# B&R Automation Studio project NAEUL004C00R13L518F00 (part 65)

#### Local.var
```iecst
(*2021-08-01*)
(**)
(*Local Action, State & Status*)
VAR
	eAct : eHermesAction := HermesActIdle;
	eStat : eHermesAction := HermesActIdle;
	eHermesAct : eHermesAction;
	eMcParamAct : eMcParamAction;
	eMainStatus : eFBStatus := Idle;
	eStatus : eFBStatus := Idle;
	eStatus1 : eFBStatus := Idle;
	eStatus2 : eFBStatus := Idle;
	eStatus3 : eFBStatus := Idle;
	udiStatus : UDINT := 0;
	udiStatus1 : UDINT := 0;
	udiStatus2 : UDINT := 0;
	udiStatus3 : UDINT := 0;
	udiStatus4 : UDINT := 0;
	udiStatus5 : UDINT;
	sStatTxt : STRING[200] := '';
	a_sStatText : ARRAY[0..50] OF STRING[200] := ['Idling','Background Starting Operations','Background Stopping Operations','Deleting Old Log File','Creating Directory','Writing Retain File','Reading Retain File','Saving Configuration',43('')];
END_VAR
(**)
(*Local Alarm*)
VAR
	tyAlmData : tyAlmDat;
	tyAlmData1 : tyAlmDat;
	tyAlmData2 : tyAlmDat;
	tyAlmData3 : tyAlmDat;
	tyAlmData4 : tyAlmDat;
	tyInfoData : tyAlmDat;
	tyInfoData1 : tyAlmDat;
	tyInfoData2 : tyAlmDat;
	tyInfoData3 : tyAlmDat;
	tyInfoData4 : tyAlmDat;
	a_tyAlmText : ARRAY[10000..10250] OF tyAlmTxt := [(sAlmText:='Invalid Ident While Creating Server',sRcyText:='Problem Occurred In The TCP/IP Connection. Check The Connection And Try To Reconnect.'),(sAlmText:='Setting Keep Alive Interval Time Error While Creating Server',sRcyText:='Unable To Establish Connection Between Machine. Check For Setting And Resume Operation.'),(sAlmText:='Setting Keep Alive Idle Time Error While Creating Server',sRcyText:='Unable To Establish Connection Between Machine. Check For Setting And Resume Operation.'),(sAlmText:='Setting Keep Alive Count Error While Creating Server',sRcyText:='Unable To Establish Connection Between Machine. Check For Setting And Resume Operation.'),(sAlmText:='Setting Keep Alive Error While Creating Server',sRcyText:='Unable To Establish Connection Between Machine. Check For Setting And Resume Operation.'),(sAlmText:='Setting Receive Buffer Error While Creating Server',sRcyText:='Unable To Establish Connection Between Machine. Check For Setting And Resume Operation.'),(sAlmText:='Setting Send Buffer Error While Creating Server',sRcyText:='Unable To Establish Connection Between Machine. Check For Setting And Resume Operation.'),(sAlmText:='Setting No Waiting Error While Creating Server',sRcyText:='Unable To Establish Connection Between Machine. Check For Setting And Resume Operation.'),(sAlmText:='TCP Open Port Error While Creating Server',sRcyText:='Problem Occurred In The TCP/IP Connection. Check The Connection And Try To Reconnect.'),(sAlmText:='Closing TCP Error While Creating Server',sRcyText:='Problem Occurred In The TCP/IP Connection. Check The Connection And Try To Reconnect.'),(sAlmText:='Invalid Ident While Listening Client',sRcyText:='There Was A Problem Connecting To The Server. The Server May Not Exist or It is Unavailable At This Time. Check The Connection and Try Again.'),(0),(sAlmText:='Supervisory Hermes Connection Lost',sRcyText:='There Was A Problem Connecting To The Server. The Server May Not Exist or It is Unavailable At This Time. Check The Connection and Try Again.'),(0),(sAlmText:='Invalid Ident While Receiving Data',sRcyText:='Problem Occurred In The TCP/IP Connection. Check The Connection And Try To Reconnect.'),(sAlmText:='TCP Receive Data Error While Receiving Data',sRcyText:='Problem Occurred In The TCP/IP Connection. Check The Connection And Try To Reconnect.'),(sAlmText:='Receive SetConfiguration While Supervisory In Not Connected State',sRcyText:='Receive Illegal Message.'),(sAlmText:='Receive GetConfiguration While Supervisory In Not Connected State',sRcyText:='Receive Illegal Message.'),(sAlmText:='Receive CurrConfiguration While Supervisory In Not Connected State',sRcyText:='Receive Illegal Message.'),(sAlmText:='Receive SendWorkOrderInfo While Supervisory In Not Connected State',sRcyText:='Receive Illegal Message.'),(sAlmText:='Receive QueryWorkOrderInfo While Supervisory In Not Connected State',sRcyText:='Receive Illegal Message.'),(sAlmText:='Receive BoardArrived While Supervisory In Not Connected State',sRcyText:='Receive Illegal Message.'),(sAlmText:='Receive BoardDeparted While Supervisory In Not Connected State',sRcyText:='Receive Illegal Message.'),2((0)),(sAlmText:='Receive BoardAvailable While Downstream In Service Description State',sRcyText:='Receive Illegal Message.'),(sAlmText:='Receive RevokeBoardAvailable While Downstream In Service Description State',sRcyText:='Receive Illegal Message.'),(sAlmText:='Receive ServiceDescription While Supervisory In Service Description State',sRcyText:='Receive Illegal Message.'),(sAlmText:='Receive SetConfiguration While Supervisory In Service Description State',sRcyText:='Receive Illegal Message.'),(sAlmText:='Receive GetConfiguration While Supervisory In Service Description State',sRcyText:='Receive Illegal Message.'),(sAlmText:='Receive CurrConfiguration While Supervisory In Service Description State',sRcyText:='Receive Illegal Message.'),(sAlmText:='Receive SendWorkOrderInfo While Supervisory In Service Description State',sRcyText:='Receive Illegal Message.'),(sAlmText:='Receive QueryWorkOrderInfo While Supervisory In Service Description State',sRcyText:='Receive Illegal Message.'),(sAlmText:='Receive BoardArrived While Supervisory In Service Description State',sRcyText:='Receive Illegal Message.'),(sAlmText:='Receive BoardDeparted While Supervisory In Service Description State',sRcyText:='Receive Illegal Message.'),4((0)),(sAlmText:='Receive ServiceDescription While Supervisory In Connected State',sRcyText:='Receive Illegal Message.'),(sAlmText:='Receive CurrConfiguration While Supervisory In Connected State',sRcyText:='Receive Illegal Message.'),(sAlmText:='Receive QueryWorkOrderInfo While Supervisory In Connected State',sRcyText:='Receive Illegal Message.'),(sAlmText:='Receive BoardArrived While Supervisory In Connected State',sRcyText:='Receive Illegal Message.'),(sAlmText:='Receive BoardDeparted While Supervisory In Connected State',sRcyText:='Receive Illegal Message.'),43((0)),(sAlmText:='SystemId Missing While Checking Service Description',sRcyText:='Missing Input Value For SystemId. Fill Up The Value And Resend.'),(sAlmText:='Version Missing While Checking Service Description',sRcyText:='Missing Input Value For Version. Fill Up The Value And Resend.'),(sAlmText:='SupportedFeatures Missing While Checking Service Description',sRcyText:='Missing Input Value For SupportedFeatures. Fill Up The Value And Resend.'),2((0)),(sAlmText:='NotificationCode Out Of Range While Checking Notification',sRcyText:='NotificationCode Does Not Fall Within The Expected Range.'),(sAlmText:='NotificationCode Missing While Checking Notification',sRcyText:='Missing Input Value For NotificationCode. Fill Up The Value And Resend.'),(sAlmText:='Severity Missing While Checking Notification',sRcyText:='Missing Input Value For Severity. Fill Up The Value And Resend.'),(sAlmText:='Description Missing While Checking Notification',sRcyText:='Missing Input Value For Description. Fill Up The Value And Resend.'),10((0)),(sAlmText:='Supervisory Service Description Interchange Time Out',sRcyText:='Timeout Expired Before Operation Completed. Reset And Resume Operation.'),4((0)),(sAlmText:='Get Directory Info Error While Deleting Old Log',sRcyText:='An Error Was Encountered While Getting Directory Info. Please Contact Nutek For A Possible Solution.'),(sAlmText:='Directory Read Error While Deleting Old Log',sRcyText:='An Error Was Encountered While Reading Directory. Please Contact Nutek For A Possible Solution.'),(sAlmText:='File Delete Error While Deleting Old Log',sRcyText:='An Error Was Encountered While Trying To Delete File. Please Contact Nutek For A Possible Solution.'),(sAlmText:='File Open Error While Reading Retain File',sRcyText:='An Error Was Encountered While Trying To Open File. Please Contact Nutek For A Possible Solution.'),(sAlmText:='File Read Error While Reading Retain File',sRcyText:='An Error Was Encountered While Trying To Read File. Please Contact Nutek For A Possible Solution.'),(sAlmText:='File Close Error While Reading Retain File',sRcyText:='An Error Was Encountered While Trying To Close File. Please Contact Nutek For A Possible Solution.'),(sAlmText:='File Open Error While Writting Retain File',sRcyText:='An Error Was Encountered While Trying To Open File. Please Contact Nutek For A Possible Solution.'),(sAlmText:='File Create Error While Writting Retain File',sRcyText:='An Error Was Encountered While Trying To Create File. Please Contact Nutek For A Possible Solution.'),(sAlmText:='File Write Error While Writting Retain File',sRcyText:='An Error Was Encountered While Trying To Write File. Please Contact Nutek For A Possible Solution.'),(sAlmText:='File Close Error While Writting Retain File',sRcyText:='An Error Was Encountered While Trying To Close File. Please Contact Nutek For A Possible Solution.'),(sAlmText:='Directory Does Not Exist While Writing Retain File',sRcyText:='The Directory Does Not Exist. Please Contact Nutek For A Possible Solution.'),(sAlmText:='Revoke Board Available Request To Send From Supervisory Hermes',sRcyText:='Sending Illegal Message.'),(sAlmText:='Stop Transport Request To Send From Supervisory Hermes',sRcyText:='Sending Illegal Message.'),(sAlmText:='Transport Finished Request To Send From Supervisory Hermes',sRcyText:='Sending Illegal Message.'),(sAlmText:='Board Available Request To Send From Supervisory Hermes',sRcyText:='Sending Illegal Message.'),6((0)),(sAlmText:='Check Alive Time Out',sRcyText:='Timeout Expired Before Operation Completed. Reset And Resume Operation.'),(sAlmText:='Waiting Check Alive Time Out',sRcyText:='Timeout Expired Before Operation Completed. Reset And Resume Operation.'),(sAlmText:='Check Alive Id Mismatch',sRcyText:='The Check Alive Id Value Does Not Match. Change The Value And Resend The Value.'),(sAlmText:='Machine Ready Request To Send From Supervisory Hermes',sRcyText:='Sending Illegal Message.'),(sAlmText:='Revoke Machine Ready Request To Send From Supervisory Hermes',sRcyText:='Sending Illegal Message.'),(sAlmText:='Start Transport Request To Send From Supervisory Hermes',sRcyText:='Sending Illegal Message.'),(sAlmText:='Set Configuration Request To Send From Supervisory Hermes',sRcyText:='Sending Illegal Message.'),(sAlmText:='Get Configuration Request To Send From Supervisory Hermes',sRcyText:='Sending Illegal Message.'),(sAlmText:='Current Configuration Request To Send From Supervisory Hermes',sRcyText:='Sending Illegal Message.'),(sAlmText:='Board Forecast Request To Send From Supervisory Hermes',sRcyText:='Sending Illegal Message.'),(sAlmText:='Query Board Info Request To Send From Supervisory Hermes',sRcyText:='Sending Illegal Message.'),(sAlmText:='Invalid Ident While Sending Data',sRcyText:='Invalid Ident Value.'),(sAlmText:='TCP Retry Send Data Error While Sending Data',sRcyText:='Problem Occurred In The TCP/IP Connection. Check The Connection And Try To Reconnect.'),(sAlmText:='TCP Send Data Error',sRcyText:='Problem Occurred In The TCP/IP Connection. Check The Connection And Try To Reconnect.'),(sAlmText:='Invalid Ident While Closing TCP',sRcyText:='Invalid Ident Value.'),(sAlmText:='Closing TCP Error',sRcyText:='Problem Occurred In The TCP/IP Connection. Check The Connection And Try To Reconnect.'),(sAlmText:='File Open Error While Writing Log',sRcyText:='An Error Was Encountered While Trying To Open File. Please Contact Nutek For A Possible Solution.'),(sAlmText:='File Create Error While Writing Log',sRcyText:='An Error Was Encountered While Trying To Create File. Please Contact Nutek For A Possible Solution.'),(sAlmText:='Get File Info Error While Writing Log',sRcyText:='An Error Was Encountered While Getting File Info. Please Contact Nutek For A Possible Solution.'),(sAlmText:='File Write Error While Writing Log',sRcyText:='An Error Was Encountered While Trying To Write File. Please Contact Nutek For A Possible Solution.'),(sAlmText:='File Close Error While Writing Log',sRcyText:='An Error Was Encountered While Trying To Close File. Please Contact Nutek For A Possible Solution.'),(sAlmText:='Directory Does Not Exist While Writing Log',sRcyText:='The Directory Does Not Exist.Please Contact Nutek For A Possible Solution.'),(sAlmText:='Invalid Ident While Closing TCP',sRcyText:='Invalid Ident Value.'),(sAlmText:='Closing TCP Error',sRcyText:='Problem Occurred In The TCP/IP Connection. Check The Connection And Try To Reconnect.'),3((0)),(sAlmText:='Send Board Info Request To Send From Supervisory Hermes',sRcyText:='Sending Illegal Message.'),(sAlmText:='Query Work Order Info Request To Send From Supervisory Hermes',sRcyText:='Sending Illegal Message.'),(sAlmText:='Send Work Order Info Request To Send From Supervisory Hermes',sRcyText:='Sending Illegal Message.'),(sAlmText:='Board Arrived Request To Send From Supervisory Hermes',sRcyText:='Sending Illegal Message.'),(sAlmText:='Board Depated Request To Send From Supervisory Hermes',sRcyText:='Sending Illegal Message.'),(sAlmText:='QueryId Mismatch While Checking SendWorkOrderInfo and QueryWorkOrderInfo',sRcyText:='The QueryId Value Does Not Match. Change The Value And Resend The Value.'),(sAlmText:='QueryId Missing While Checking Send Work Order Info',sRcyText:='Missing Input Value For QueryId. Fill Up The Value And Resend.'),20((0)),(sAlmText:='File Open Error While Writing Config File',sRcyText:='An Error Was Encountered While Trying To Open File. Please Contact Nutek For A Possible Solution.'),(sAlmText:='File Create Error While Writing Config File',sRcyText:='An Error Was Encountered While Trying To Create File. Please Contact Nutek For A Possible Solution.'),(sAlmText:='File Write Error While Writing Config File',sRcyText:='An Error Was Encountered While Trying To Write File. Please Contact Nutek For A Possible Solution.'),(sAlmText:='File Close Error While Writing Config File',sRcyText:='An Error Was Encountered While Trying To Close File. Please Contact Nutek For A Possible Solution.'),(sAlmText:='Directory Does Not Exist While Writing Config File',sRcyText:='The Directory Does Not Exist. Please Contact Nutek For A Possible Solution.'),9((0)),(sAlmText:='File Open Error While Reading Loader Work Order Retain File',sRcyText:='An Error Was Encountered While Trying To Open File. Please Contact Nutek For A Possible Solution.'),(sAlmText:='File Read Error While Reading Loader Work Order Retain File',sRcyText:='An Error Was Encountered While Trying To Read File. Please Contact Nutek For A Possible Solution.'),(sAlmText:='File Close Error While Reading Loader Work Order Retain File',sRcyText:='An Error Was Encountered While Trying To Close File. Please Contact Nutek For A Possible Solution.'),(sAlmText:='File Open Error While WrittingLoader Work Order  Retain File',sRcyText:='An Error Was Encountered While Trying To Open File. Please Contact Nutek For A Possible Solution.'),(sAlmText:='File Create Error While Writting Loader Work Order Retain File',sRcyText:='An Error Was Encountered While Trying To Create File. Please Contact Nutek For A Possible Solution.'),(sAlmText:='File Write Error While Writting Loader Work Order Retain File',sRcyText:='An Error Was Encountered While Trying To Write File. Please Contact Nutek For A Possible Solution.'),(sAlmText:='File Close Error While Writting Loader Work Order  Retain File',sRcyText:='An Error Was Encountered While Trying To Close File. Please Contact Nutek For A Possible Solution.'),(sAlmText:='Directory Does Not Exist While Loader Work Order Writing Retain File',sRcyText:='The Directory Does Not Exist. Please Contact Nutek For A Possible Solution.'),(sAlmText:='File Open Error While Reading Loader Loaded Work Order Retain File',sRcyText:='An Error Was Encountered While Trying To Open File. Please Contact Nutek For A Possible Solution.'),(sAlmText:='File Read Error While Reading Loader Loaded Work Order Retain File',sRcyText:='An Error Was Encountered While Trying To Read File. Please Contact Nutek For A Possible Solution.'),(sAlmText:='File Close Error While Reading Loader Loaded Work Order Retain File',sRcyText:='An Error Was Encountered While Trying To Close File. Please Contact Nutek For A Possible Solution.'),(sAlmText:='File Open Error While Writting Loader Loaded Work Order Retain File',sRcyText:='An Error Was Encountered While Trying To Open File. Please Contact Nutek For A Possible Solution.'),(sAlmText:='File Create Error While Writting Loaded Work Order Retain File',sRcyText:='An Error Was Encountered While Trying To Create File. Please Contact Nutek For A Possible Solution.'),(sAlmText:='File Write Error While Writting Loader Loaded Work Order Retain File',sRcyText:='An Error Was Encountered While Trying To Write File. Please Contact Nutek For A Possible Solution.'),(sAlmText:='File Close Error While Writting Loader Loaded Work Order Retain File',sRcyText:='An Error Was Encountered While Trying To Close File. Please Contact Nutek For A Possible Solution.'),(sAlmText:='Directory Does Not Exist While Writing Loader Loaded Work Order Retain File',sRcyText:='The Directory Does Not Exist. Please Contact Nutek For A Possible Solution.'),(sAlmText:='File Open Error While Reading Bypass Work Order Retain File',sRcyText:='An Error Was Encountered While Trying To Open File. Please Contact Nutek For A Possible Solution.'),(sAlmText:='File Read Error While Reading Bypass  Work Order Retain File',sRcyText:='An Error Was Encountered While Trying To Read File. Please Contact Nutek For A Possible Solution.'),(sAlmText:='File Close Error While Reading Bypass Work Order Retain File',sRcyText:='An Error Was Encountered While Trying To Close File. Please Contact Nutek For A Possible Solution.'),(sAlmText:='File Open Error While Writting Bypass Work Order Retain File',sRcyText:='An Error Was Encountered While Trying To Open File. Please Contact Nutek For A Possible Solution.'),(sAlmText:='File Create Error While Writting Bypass  Work Order Retain File',sRcyText:='An Error Was Encountered While Trying To Create File. Please Contact Nutek For A Possible Solution.'),(sAlmText:='File Write Error While Writting Bypass  Work Order Retain File',sRcyText:='An Error Was Encountered While Trying To Write File. Please Contact Nutek For A Possible Solution.'),(sAlmText:='File Close Error While Writting Bypass  Work Order Retain File',sRcyText:='An Error Was Encountered While Trying To Close File. Please Contact Nutek For A Possible Solution.'),(sAlmText:='Directory Does Not Exist While Writing Bypass  Work Order Retain File',sRcyText:='The Directory Does Not Exist. Please Contact Nutek For A Possible Solution.'),0,26((0))];
END_VAR
(**)
(*Local Output*)
VAR
	bConnected : BOOL;
	bTest : BOOL;
	bTest1 : BOOL;
	bTest2 : BOOL;
	bHandshakeDone : BOOL;
	sInternalSnd : STRING[65535];
	bFileNotFound : BOOL := FALSE;
	bWriteConfig : BOOL := FALSE;
	bUpdateUIData : BOOL := FALSE;
END_VAR
(**)
(*Local Input*)
VAR
	udiRstErr : UDINT := 0;
	bPrep : BOOL := TRUE;
	bEn : BOOL := TRUE;
	bDis : BOOL := FALSE;
	tyParam : tyHermesSvyParam;
	sIPAddr : STRING[15] := '192.168.0.100';
	a_usiMacAddr : ARRAY[0..5] OF USINT := [6(0)];
	tyDTStructure : DTStructure := (year:=2020,month:=11,day:=05,wday:=05,hour:=21,minute:=28,second:=30,millisec:=123,microsec:=456);
	dtCurrDT : DATE_AND_TIME := DT#2019-02-23-12:30:50;
	sMcId : STRING[80] := '';
	sMagazineId : STRING[80] := '';
	iSlotId : INT;
	sBarcode : STRING[254] := '';
	eBoardTransfer1 : eHermesBoardTransfer := HermesTransferred;
	eBoardTransfer2 : eHermesBoardTransfer := HermesTransferred;
	eBoardTransfer3 : eHermesBoardTransfer := HermesTransferred;
	eBoardTransfer4 : eHermesBoardTransfer := HermesTransferred;
	sVersion : STRING[7] := '1.3';
	sWorkOrderId : STRING[80] := '';
	sBatchId : STRING[80] := '';
	sRecipeNm : STRING[254] := '';
	udiSndBffrSize : UDINT := 65536;
	udiRcvBffrSize : UDINT := 65536;
	udiAliveIdleTimeInSec : UDINT := 5;
	tConnTimeOut : TIME := T#30s;
	diTransferInTO : DINT := 30000;
	bNewBrdAvl : BOOL := FALSE;
	bOpsRun : BOOL := FALSE;
	udiFileKeepDay : UDINT := 30;
	sConfigFileName : STRING[80] := 'SvyHermes.dat';
	sProgNm : STRING[15] := 'SvyHermes';
	sRetainFileName : STRING[80] := 'WorkOrder.dat';
	sRetainFileName1 : STRING[80] := 'LoaderSendWorkOrder.dat';
	sRetainFileName2 : STRING[80] := 'LoaderLoadedSendWorkOrder.dat';
	sRetainFileName3 : STRING[80] := 'BypassSendWorkOrder.dat';
	bNtSettingsLoadDone : BOOL := TRUE;
	bSvyPrep : BOOL := FALSE;
	bSvyEn : BOOL := FALSE;
	sInfoMsg : STRING[200];
	sInfoMsg1 : STRING[200];
	sInfoMsg2 : STRING[200];
	sInfoMsg3 : STRING[200];
	sInfoMsg4 : STRING[200];
	bEndSen : BOOL := FALSE;
	tyHermesCurrConfiguration : tyHermesConfiguration;
	bQueryWorkOrderInfo : BOOL;
	bAcceptCondition : BOOL;
	bAllZonesEmpty : BOOL;
	bDeleteWorkOrder : BOOL;
	bFirstMcIntheLine : BOOL;
	bUSHermesStopTransportSnd1 : BOOL;
	bUSHermesStopTransportSnd2 : BOOL;
	bUSHermesStopTransportSnd3 : BOOL;
	bUSHermesStopTransportSnd4 : BOOL;
	bDSHermesTransportFinishedSnd1 : BOOL;
	bDSHermesTransportFinishedSnd2 : BOOL;
	bDSHermesTransportFinishedSnd3 : BOOL;
	bDSHermesTransportFinishedSnd4 : BOOL;
	tyUSHermesBoardArrivedData1 : tyHermesBoardAvailable;
	tyUSHermesBoardArrivedData2 : tyHermesBoardAvailable;
	tyUSHermesBoardArrivedData3 : tyHermesBoardAvailable;
	tyUSHermesBoardArrivedData4 : tyHermesBoardAvailable;
	tyDSHermesBoardDepartedData1 : tyHermesBoardAvailable;
	tyDSHermesBoardDepartedData2 : tyHermesBoardAvailable;
	tyDSHermesBoardDepartedData3 : tyHermesBoardAvailable;
	tyDSHermesBoardDepartedData4 : tyHermesBoardAvailable;
	bInternalUse : BOOL;
	sInternalRcv : STRING[65535];
END_VAR
(**)
(*Local*)
VAR
	bRstErr : BOOL;
	udiRstErrOld : UDINT;
	bInitDone : BOOL;
	bInitialDone : BOOL;
	bRun : BOOL;
	bStop : BOOL;
	bRstConnection : BOOL;
	bRstState : BOOL;
	bRcvWorkOrderInfo1 : BOOL;
	bRcvWorkOrderInfo2 : BOOL;
	bRcvWorkOrderInfo3 : BOOL;
	bRcvBypassWorkOrderInfo2 : BOOL;
	bRstWorkOrderInfo : BOOL;
	bFoundIndexUS1 : BOOL;
	bFoundIndexUS2 : BOOL;
	bFoundIndexUS3 : BOOL;
	bFoundIndexUS4 : BOOL;
	bFoundIndexDS1 : BOOL;
	bFoundIndexDS2 : BOOL;
	bFoundIndexDS3 : BOOL;
	bFoundIndexDS4 : BOOL;
	udiFoundIndexUS1 : UDINT;
	udiFoundIndexUS2 : UDINT;
	udiFoundIndexUS3 : UDINT;
	udiFoundIndexUS4 : UDINT;
	udiFoundIndexDS1 : UDINT;
	udiFoundIndexDS2 : UDINT;
	udiFoundIndexDS3 : UDINT;
	udiFoundIndexDS4 : UDINT;
	k : UDINT := 0;
	kk : UDINT := 0;
	j : INT := 1;
	jj : INT := 2;
	jjj : INT := 3;
	jjjj : INT := 4;
	udiSvrIdent : UDINT;
	udiClntIdent : UDINT;
	udiClntIdentExtra : UDINT;
	udiXMLTableWriteIdx : UDINT;
	udiMsgSendBffr : UDINT;
	udiSndMsgLen : UDINT;
	sSnd : STRING[65535];
	sRcv : STRING[65535];
	a_tyXMLTableDataRcv : ARRAY[0..200] OF tyXMLTableDat;
	a_tyXMLTableDataSnd : ARRAY[0..200] OF tyXMLTableDat;
	a_eMsgSend : ARRAY[0..50] OF eHermesMsgType;
	tyMsgTypeRcv : tyHermesMsgType;
	tyCheckAliveSnd : tyHermesCheckAlive;
	tyCheckAlivePingSnd : tyHermesCheckAlive;
	tyCheckAlivePongSnd : tyHermesCheckAlive;
	tyCheckAliveRcv : tyHermesCheckAlive;
	tyCheckAlivePingRcv : tyHermesCheckAlive;
	tyCheckAlivePongRcv : tyHermesCheckAlive;
	tyServiceDescriptionRcv : tyHermesServiceDescription;
	tySServiceDescriptionSnd : tyHermesSServiceDescription;
	tySServiceDescriptionRcv : tyHermesSServiceDescription;
	tyNotificationSnd : tyHermesNotification;
	tyNotificationRcv : tyHermesNotification;
	tyBoardAvailableRcv : tyHermesBoardAvailable;
	tyMachineReady : tyHermesMachineReady;
	tyStartTransport : tyHermesStartTransport;
	tyStopTransport : tyHermesStopTransport;
	tyTransportFinished : tyHermesTransportFinished;
	tySetConfiguration : tyHermesSetConfiguration;
	tySetConfigurationRcv : tyHermesSetConfiguration;
	tySetConfigurationModified : tyHermesSetConfiguration;
	tyCurrentConfigurationRcv : tyHermesCurrentConfiguration;
	tyCurrentConfigurationSnd : tyHermesCurrentConfiguration;
	tyBoardForecast : tyHermesBoardForecast;
	tyBoardArrivedRcv : tyHermesBoardArrived;
	tyBoardArrived1 : tyHermesBoardArrived;
	tyBoardArrived2 : tyHermesBoardArrived;
	tyBoardArrived3 : tyHermesBoardArrived;
	tyBoardArrived4 : tyHermesBoardArrived;
	tyBoardDepartedRcv : tyHermesBoardDeparted;
	tyBoardDeparted1 : tyHermesBoardDeparted;
	tyBoardDeparted2 : tyHermesBoardDeparted;
	tyBoardDeparted3 : tyHermesBoardDeparted;
	tyBoardDeparted4 : tyHermesBoardDeparted;
	tyQueryBoardInfo : tyHermesQueryBoardInfo;
	tySendBoardInfo : tyHermesSendBoardInfo;
	tyQueryWorkOrderInfo : tyHermesQueryWorkOrderInfo; (*Query For Loader Mode*)
	tyQueryBypassWorkOrderInfo : tyHermesQueryWorkOrderInfo; (*Query For Bypass mode*)
	tyReplyWorkOrderInfo : tyHermesReplyWorkOrderInfo;
	tySendWorkOrderInfoAcc : tyHermesSendWorkOrderInfo;
	tySendBypassWorkOrderInfoAcc : tyHermesSendWorkOrderInfo;
	tySendWorkOrderInfoRcv : tyHermesSendWorkOrderInfo;
	tyDummySendWorkOrderInfoRcv : tyHermesSendWorkOrderInfo;
	tySendWorkOrderInfoNewAcc : tyHermesSendWorkOrderInfo;
	fbCreateSvr : fbTCPCreateSvr;
	fbListen : fbTCPListen;
	fbRcv : fbTCPRcv;
	fbSend : fbTCPSnd;
	fbCloseSvr : fbTCPClose;
	fbCloseClnt : fbTCPClose;
	fbParseXMLTable : fbHermesParseXMLTable;
	fbCheckAlive : fbHermesCheckAlive;
	fbCheckAliveSendPing : fbHermesCheckAliveSendPing;
	fbCheckAliveRcvPing : fbHermesCheckAliveRcvPing;
	fbSequenceSvy : fbHermesSequenceSvy;
	fbSequenceTO : fbHermesSequenceSvyTO;
	eStatOld : eHermesAction := HermesActIdle;
	tyParamOld : tyHermesSvyParam;
	udiLogCntr : UDINT := 1;
	udiWriteLogCntr : UDINT := 1;
	a_sLogList : ARRAY[1..10] OF STRING[65535];
	sDT : STRING[80];
	dtCurrDTTemp : DATE_AND_TIME;
	fbFileAppend1 : fbFileFullAppend;
	fbFileOldDel1 : fbFileOldDel;
	fbFileRead1 : fbFileFullRead;
	fbFileWrite1 : fbFileFullWrite;
	fbFileRead2 : fbFileFullRead;
	fbFileWrite2 : fbFileFullWrite;
	fbFileRead3 : fbFileFullRead;
	fbFileWrite3 : fbFileFullWrite;
	fbFileRead4 : fbFileFullRead;
	fbFileWrite4 : fbFileFullWrite;
	fbDelayTm : TON;
	fbDelayTm1 : TON;
	fbParseBrdAvlExternal : fbHermesParseXMLTable;
	tyDsInternalBoardDeparted : {REDUND_UNREPLICABLE} tyHermesBoardAvailable;
	rThickness : REAL;
	rConveyorSpeed : REAL;
	rTopClearanceHeight : REAL;
	rBottomClearanceHeight : REAL;
	rWeight : REAL;
	udiTargetAddress : UDINT := 0;
	udiTargetAddress1 : UDINT := 0;
	udiSizeAddress : UDINT := 0;
	udiSizeAddress1 : UDINT := 0;
	udiRetainDataAddr : UDINT;
	udiRetainDataLen : UDINT;
	udiLoaderRetainDataAddr0 : UDINT;
	udiLoaderRetainDataLen0 : UDINT;
	udiLoaderRetainDataAddr1 : UDINT;
	udiLoaderRetainDataLen1 : UDINT;
	udiBypassRetainDataAddr0 : UDINT;
	udiBypassRetainDataLen0 : UDINT;
	tyHermesBARcv : tyHermesBoardAvailable;
	tyHermesBFRcv : tyHermesBoardForecast;
	bOpsConvWaitForTopUpBrd : BOOL;
	diReqWidthInUM : DINT;
	diReqLoaderWidthInUM : DINT;
	iWriteLogStep : INT := 0;
	bDIPresentSen : BOOL;
	bUITopUpBrdRdy : BOOL;
	bOpsConvStepAllwTopUpBrd : BOOL;
	bOpsConvTopUpBrdReq : BOOL;
	bLinkStepStackMode : BOOL;
	udiModuleNum : UDINT := 6761;
	bTransportFinish1 : BOOL;
	bTransportFinish2 : BOOL;
	bTransportFinish3 : BOOL;
END_VAR
```

#### Act_Alarm.st
```iecst
(** 2021-08-01 **)
ACTION Act_Alarm: //General

	//Error
	IF EDGEPOS(eStatus = Error) THEN

		tyAlmData.sProgNm		:= p_sProgNm;
		tyAlmData.udiCode		:= udiStatus;
		tyAlmData.eSeverity		:= AlmSeverityError;
		tyAlmData.udiRunTime	:= tyAlmData.udiRunTime + 1;
		tyAlmData.bAlm			:= TRUE;
		tyAlmData.udiModuleNum  := udiModuleNum;
		g_sSvyHermesProgNm		:= p_sProgNm;
		//Get Error Message
		IF tyAlmData.udiCode < 10000 OR tyAlmData.udiCode > 10199 THEN
			tyAlmData.sAlmMsg	:= 'Unknown';
			tyAlmData.sRcyMsg	:= 'Unknown';
		ELSE
			tyAlmData.sAlmMsg	:= a_tyAlmText[tyAlmData.udiCode].sAlmText;
			tyAlmData.sRcyMsg	:= a_tyAlmText[tyAlmData.udiCode].sRcyText;
		END_IF

		sStatTxt	:= tyAlmData.sAlmMsg;

	ELSIF bRstErr AND (tyAlmData.udiCode <> 0) THEN

		tyAlmData.udiCode	:= 0;
		tyAlmData.eSeverity	:= AlmSeverityNA;
		tyAlmData.sAlmMsg	:= '';
		tyAlmData.sRcyMsg	:= '';
		tyAlmData.bAlm			:= FALSE;
		sStatTxt	:= a_sStatText[eStat];

	END_IF

END_ACTION
```

#### Act_Alarm1.st
```iecst
(** 2021-08-01 **)
ACTION Act_Alarm1:

	//Error
	IF EDGEPOS(eStatus1 = Error) THEN

		tyAlmData1.sProgNm		:= p_sProgNm;
		tyAlmData1.udiCode		:= udiStatus1;
		tyAlmData1.eSeverity	:= AlmSeverityError;
		tyAlmData1.udiRunTime	:= tyAlmData1.udiRunTime + 1;
		tyAlmData1.bAlm			:= TRUE;
		tyAlmData1.udiModuleNum  := udiModuleNum;
		g_sSvyHermesProgNm		:= p_sProgNm;
		//Get Error Message
		IF tyAlmData1.udiCode < 10000 OR tyAlmData1.udiCode > 10199 THEN
			tyAlmData1.sAlmMsg	:= 'Unknown';
			tyAlmData1.sRcyMsg	:= 'Unknown';
		ELSE
			tyAlmData1.sAlmMsg	:= a_tyAlmText[tyAlmData1.udiCode].sAlmText;
			tyAlmData1.sRcyMsg	:= a_tyAlmText[tyAlmData1.udiCode].sRcyText;
		END_IF

		sStatTxt	:= tyAlmData1.sAlmMsg;

	ELSIF bRstErr AND (tyAlmData1.udiCode <> 0) THEN

		tyAlmData1.udiCode		:= 0;
		tyAlmData1.eSeverity	:= AlmSeverityNA;
		tyAlmData1.sAlmMsg		:= '';
		tyAlmData1.sRcyMsg		:= '';
		tyAlmData1.bAlm			:= FALSE;
		sStatTxt	:= a_sStatText[eStat];

	END_IF

END_ACTION
```

#### Act_Alarm2.st
```iecst
(** 2021-08-01 **)
ACTION Act_Alarm2:

	//Error
	IF EDGEPOS(eStatus2 = Error) THEN

		tyAlmData2.sProgNm		:= p_sProgNm;
		tyAlmData2.udiCode		:= udiStatus2;
		tyAlmData2.eSeverity	:= AlmSeverityError;
		tyAlmData2.udiRunTime	:= tyAlmData2.udiRunTime + 1;
		tyAlmData2.bAlm			:= TRUE;
		tyAlmData2.udiModuleNum  := udiModuleNum;
		g_sSvyHermesProgNm		:= p_sProgNm;
		//Get Error Message
		IF tyAlmData2.udiCode < 10000 OR tyAlmData2.udiCode > 10199 THEN
			tyAlmData2.sAlmMsg	:= 'Unknown';
			tyAlmData2.sRcyMsg	:= 'Unknown';
		ELSE
			tyAlmData2.sAlmMsg	:= a_tyAlmText[tyAlmData2.udiCode].sAlmText;
			tyAlmData2.sRcyMsg	:= a_tyAlmText[tyAlmData2.udiCode].sRcyText;
		END_IF

		sStatTxt	:= tyAlmData2.sAlmMsg;

	ELSIF bRstErr AND (tyAlmData2.udiCode <> 0) THEN

		tyAlmData2.udiCode		:= 0;
		tyAlmData2.eSeverity	:= AlmSeverityNA;
		tyAlmData2.sAlmMsg		:= '';
		tyAlmData2.sRcyMsg		:= '';
		tyAlmData2.bAlm			:= FALSE;
		sStatTxt	:= a_sStatText[eStat];

	END_IF

END_ACTION
```

#### Act_Alarm3.st
```iecst
(** 2021-08-01 **)
ACTION Act_Alarm3: //fbFileAppend1 Error

	//Error
	IF EDGEPOS(eStatus3 = Error) THEN

		tyAlmData3.sProgNm		:= p_sProgNm;
		tyAlmData3.udiCode		:= udiStatus3;
		tyAlmData3.eSeverity	:= AlmSeverityError;
		tyAlmData3.udiRunTime	:= tyAlmData3.udiRunTime + 1;
		tyAlmData3.bAlm			:= TRUE;
		tyAlmData3.udiModuleNum  := udiModuleNum;
		g_sSvyHermesProgNm		:= p_sProgNm;
		//Get Error Message
		IF tyAlmData3.udiCode < 10000 OR tyAlmData3.udiCode > 10199 THEN
			tyAlmData3.sAlmMsg	:= 'Unknown';
			tyAlmData3.sRcyMsg	:= 'Unknown';
		ELSE
			tyAlmData3.sAlmMsg	:= a_tyAlmText[tyAlmData3.udiCode].sAlmText;
			tyAlmData3.sRcyMsg	:= a_tyAlmText[tyAlmData3.udiCode].sRcyText;
		END_IF

		sStatTxt	:= tyAlmData3.sAlmMsg;

	ELSIF bRstErr AND (tyAlmData3.udiCode <> 0) THEN

		tyAlmData3.udiCode		:= 0;
		tyAlmData3.eSeverity	:= AlmSeverityNA;
		tyAlmData3.sAlmMsg		:= '';
		tyAlmData3.sRcyMsg		:= '';
		tyAlmData3.bAlm			:= FALSE;
		sStatTxt	:= a_sStatText[eStat];

	END_IF

END_ACTION
```

#### Act_Alarm4.st
```iecst
(** 2021-08-01 **)
ACTION Act_Alarm4: //Not Connected Warning

	//Warning
	IF ((bConnected = FALSE) AND (p_bSvyEn)) THEN

		tyAlmData4.sProgNm		:= p_sProgNm;
		tyAlmData4.udiCode		:= udiStatus4;
		tyAlmData4.eSeverity	:= AlmSeverityWarning;
		tyAlmData4.udiRunTime	:= tyAlmData4.udiRunTime + 1;
		tyAlmData4.bWarning			:= TRUE;
		tyAlmData4.udiModuleNum  := udiModuleNum;
		g_sSvyHermesProgNm		:= p_sProgNm;
		//Get Warning Message
		IF tyAlmData4.udiCode < 10000 OR tyAlmData4.udiCode > 10199 THEN
			tyAlmData4.sAlmMsg	:= 'Unknown';
			tyAlmData4.sRcyMsg	:= 'Unknown';
		ELSE
			tyAlmData4.sAlmMsg	:= a_tyAlmText[tyAlmData4.udiCode].sAlmText;
			tyAlmData4.sRcyMsg	:= a_tyAlmText[tyAlmData4.udiCode].sRcyText;
		END_IF

		sStatTxt	:= tyAlmData4.sAlmMsg;

	ELSIF (bConnected AND (tyAlmData4.udiCode <> 0)) OR (p_bSvyEn = FALSE) THEN

		tyAlmData4.udiCode		:= 0;
		tyAlmData4.eSeverity	:= AlmSeverityNA;
		tyAlmData4.sAlmMsg		:= '';
		tyAlmData4.sRcyMsg		:= '';
		tyAlmData4.bWarning			:= FALSE;
		sStatTxt	:= a_sStatText[eStat];

	END_IF

END_ACTION
```

#### Act_Background.st
```iecst
(** 2021-08-01 **)
ACTION Act_Background:

	IF bRun = TRUE THEN
		IF udiSvrIdent = 0 THEN
			IF p_bInternalUse = FALSE THEN
				Act_Background_TCPCreateSvr;

				tyParamOld	:= p_tyParam;
			ELSE
				udiSvrIdent	:= 1;
			END_IF

		ELSE
			IF bRstConnection = FALSE THEN

				Act_Background_ChgConfig;

				IF udiClntIdent = 0 THEN
					IF p_bInternalUse = FALSE THEN
						Act_Background_TCPListen;
					ELSE
						udiClntIdent	:= 1;
					END_IF

				ELSE
					Act_Background_TCPRcv;

					Act_Background_NotificationRcv;

					Act_Background_IllegalMsg;
					Act_Background_ChkParamRcv;
					Act_Background_CmpParamRcv;
					Act_Background_UpdtConfig;

					IF bHandshakeDone = TRUE THEN
						IF (p_tyParam.tSndAlive <> T#0s) AND (p_tyParam.tRcvAlive <> T#0s) THEN
							IF tySServiceDescriptionRcv.tyData.tySupportedFeatures.bFeatureCheckAliveResponse = TRUE AND p_tyParam.bFeatureCheckAliveResponse = TRUE THEN
								Act_Background_ChkAliveSendPing;
								Act_Background_ChkAliveRcvPing;
							ELSE
								Act_Background_ChkAlive;
							END_IF
						ELSE
							fbCheckAlive(bEn := FALSE);
							fbCheckAliveSendPing(bEn := FALSE);
							fbCheckAliveRcvPing(bEn := FALSE);
						END_IF
					END_IF

					Act_Background_Sequence;
					Act_Background_SequenceTO;
					Act_Background_Err;

					IF tySServiceDescriptionRcv.tyAvl.tySupportedFeatures.bFeatureSendWorkOrderInfo = TRUE AND p_tyParam.bFeatureQueryWorkOrderInfo AND bHandshakeDone THEN
						Act_Background_QueryWorkOrderInfo;
					END_IF

					Act_Background_SendBoardArrivedLane1;
					Act_Background_SendBoardArrivedLane2;
					Act_Background_SendBoardArrivedLane3;
					Act_Background_SendBoardArrivedLane4;
					Act_Background_SendBoardDepartedLane1;
					Act_Background_SendBoardDepartedLane2;
					Act_Background_SendBoardDepartedLane3;
					Act_Background_SendBoardDepartedLane4;
					Act_Background_TCPSend;

					Act_Background_Log;

				END_IF

			ELSE
				IF udiClntIdent <> 0 THEN
					Act_Background_TCPCloseClnt;
				ELSE
					IF udiSvrIdent <> 0 THEN
						Act_Background_TCPCloseSvr;
					END_IF
				END_IF

			END_IF

			//Second Client Connected
			IF udiClntIdentExtra = 0 THEN

			ELSE

			END_IF

		END_IF

		Act_Background_Stop;

	END_IF

	IF EDGENEG(bRun) OR EDGENEG(udiSvrIdent = 0) THEN
		//Reset
		fbCreateSvr(bEn := FALSE);
	END_IF

	IF EDGENEG(bRun) OR EDGENEG(udiClntIdent = 0) THEN
		//Reset
		fbListen(bEn := FALSE);

		bConnected	:= bRun;
	END_IF

	IF EDGENEG(bRun) OR EDGENEG(udiSvrIdent <> 0) OR EDGENEG(udiClntIdent <> 0) THEN
		fbRcv(bEn := FALSE);
		fbSequenceSvy(bEn := FALSE);
		fbSequenceTO(bEn := FALSE);
		fbCheckAlive(bEn := FALSE);
		fbCheckAliveSendPing(bEn := FALSE);
		fbCheckAliveRcvPing(bEn := FALSE);
		fbSend(bEn := FALSE);

		fbFileAppend1(bEn := FALSE);
		iWriteLogStep	:= 0;

		bConnected		:= FALSE;
		bHandshakeDone	:= FALSE;
		bRstState		:= FALSE;

		memset(ADR(tyMsgTypeRcv) , 0 , SIZEOF(tyMsgTypeRcv));
		memset(ADR(a_eMsgSend) , 0 , SIZEOF(a_eMsgSend));
		udiMsgSendBffr	:= 0;
	END_IF

	IF EDGENEG(bRun) OR EDGENEG(udiSvrIdent <> 0) THEN
		bRstConnection	:= FALSE;
		fbCloseSvr(bEn := FALSE);
	END_IF

	IF EDGENEG(bRun) OR EDGENEG(udiClntIdent <> 0) THEN
		fbCloseClnt(bEn := FALSE);
	END_IF

	//Reset Error
	IF (eStatus1 = Error) AND bRstErr THEN
		eStatus1	:= Idle;
		udiStatus1	:= 0;

		fbCreateSvr(bEn := FALSE);
		fbListen(bEn := FALSE);
		fbRcv(bEn := FALSE);
		fbSequenceSvy(bEn := FALSE);
		fbSend(bEn := FALSE);
		fbCloseSvr(bEn := FALSE);
		fbCloseClnt(bEn := FALSE);
		fbCheckAlive(bEn := FALSE);
		fbCheckAliveSendPing(bEn := FALSE);
		fbCheckAliveRcvPing(bEn := FALSE);
		fbSequenceTO(bEn := FALSE);

		fbFileAppend1(bEn := FALSE);
		iWriteLogStep	:= 0;

		bConnected		:= FALSE;
		bHandshakeDone	:= FALSE;
		bRstConnection	:= FALSE;
		bRstState		:= FALSE;

		memset(ADR(tyMsgTypeRcv) , 0 , SIZEOF(tyMsgTypeRcv));
		memset(ADR(a_eMsgSend) , 0 , SIZEOF(a_eMsgSend));
		udiMsgSendBffr	:= 0;
	END_IF

	IF (eStatus2 = Error) AND bRstErr THEN
		eStatus2	:= Idle;
		udiStatus2	:= 0;

		fbSequenceTO(bEn := FALSE);

	END_IF

	IF (eStatus3 = Error) AND bRstErr THEN
		eStatus3	:= Idle;
		udiStatus3	:= 0;

		fbFileAppend1(bEn := FALSE);
		iWriteLogStep	:= 0;
	END_IF

END_ACTION
```

#### Act_Background_CmpParamRcv.st
```iecst
(** 2021-08-01 **)
ACTION Act_Background_CmpParamRcv:

	IF eStatus2 <> Error THEN

		IF tySServiceDescriptionRcv.tyAvl.tySupportedFeatures.bFeatureSendWorkOrderInfo = TRUE AND p_tyParam.bFeatureQueryWorkOrderInfo THEN
				                                                                          //ADD
			IF tyMsgTypeRcv.bSendWorkOrderInfo = TRUE AND (p_bQueryWorkOrderInfo OR tyQueryWorkOrderInfo.tyAvl.bQueryId) THEN
				udiStatus2	:= fHermesChkParamSWQW(tySendWorkOrderInfoRcv , tyQueryWorkOrderInfo);
				udiStatus5  := fHermesChkParamSWBQW(tySendWorkOrderInfoRcv , tyQueryBypassWorkOrderInfo);	          //ADD

				IF udiStatus2 <> 0 AND udiStatus5 <> 0 THEN
					eStatus2	:= Error;

					IF udiStatus2 = 2767 THEN
						udiStatus2	:= 10164;	//QueryId Mismatch While Checking SendWorkOrderId & QueryWorkOrderId
					ELSIF udiStatus5 = 2767  THEN
						udiStatus2	:= 10164;	//QueryId Mismatch While Checking SendWorkOrderId & QueryWorkOrderId
					ELSIF udiStatus2 = 2768 THEN
						udiStatus2	:= 10165;	//QueryId Missing While Checking SendWorkOrderId & QueryWorkOrderId
					ELSIF udiStatus5 = 2768 THEN
						udiStatus2	:= 10165;	//QueryId Missing While Checking SendWorkOrderId & QueryWorkOrderId
					END_IF

					fHermesAddOneMsgSend(ADR(a_eMsgSend) , ADR(udiMsgSendBffr) , HermesMsgTypeNotification);

					tyNotificationSnd.tyAvl.bSeverity			:= TRUE;
					tyNotificationSnd.tyAvl.bNotificationCode	:= TRUE;
					tyNotificationSnd.tyAvl.bDescription		:= TRUE;
					tyNotificationSnd.tyData.eSeverity			:= HermesSeverityError;
					tyNotificationSnd.tyData.iNotificationCode	:= UDINT_TO_INT(udiStatus2);
					tyNotificationSnd.tyData.sDescription		:= a_tyAlmText[udiStatus2].sAlmText;

					tyMsgTypeRcv.bSendWorkOrderInfo := FALSE; //reset, else latching
				END_IF
			END_IF
		END_IF
	END_IF

		END_ACTION
```

#### Act_Background_ProcessData.st
```iecst
(** 2021-08-01 **)
ACTION Act_Background_ProcessData:

	//Write Config into "Hermes"
	fbDelayTm(IN := bWriteConfig, PT := T#0.5S); //Small Delay 0.5s to let Hermes take the Data, before WriteConfig

	IF fbDelayTm.Q THEN

		eHermesAct := HermesActWriteConfig;
		eMcParamAct := McParamActWrite;

		IF p_eHermesStatus = Done AND p_eHermesStat = HermesActWriteConfig AND p_eMcParamStat = McParamActWrite AND p_eMcParamStatus = Done THEN

		eMcParamAct     := McParamActIdle;
	   	eHermesAct		:= HermesActIdle;
		bWriteConfig    := FALSE;
		bUpdateUIData   := TRUE;
		fbDelayTm(IN := FALSE);
		tyInfoData.sProgNm		:= p_sProgNm;
		tyInfoData.udiCode		:= 10000;
		tyInfoData.eSeverity	:= AlmSeverityInfo;
		tyInfoData.sAlmMsg		:= p_sInfoMsg;

	    ELSIF  (p_eHermesStatus = Error AND p_eHermesStat = HermesActWriteConfig) OR (p_eMcParamStat = McParamActWrite AND p_eMcParamStatus = Error)  THEN

			eMcParamAct     := McParamActIdle;
		    eHermesAct		:= HermesActIdle;
		    bWriteConfig    := FALSE;
		    bUpdateUIData   := FALSE;
			fbDelayTm(IN := FALSE);

			fHermesAddOneMsgSend(ADR(a_eMsgSend) , ADR(udiMsgSendBffr) , HermesMsgTypeNotification);

			udiStatus2 := 10199; //SetConfiguration Failed, Please Send Again
			tyNotificationSnd.tyAvl.bSeverity			:= TRUE;
			tyNotificationSnd.tyAvl.bNotificationCode	:= TRUE;
			tyNotificationSnd.tyAvl.bDescription		:= TRUE;
			tyNotificationSnd.tyData.eSeverity			:= HermesSeverityFatalError;
			tyNotificationSnd.tyData.iNotificationCode	:= UDINT_TO_INT(udiStatus2);
			tyNotificationSnd.tyData.sDescription		:= a_tyAlmText[udiStatus2].sAlmText;

		END_IF
	END_IF

	//Update UI
	IF bUpdateUIData THEN
		tyInfoData.sProgNm		:= p_sProgNm;
		tyInfoData.udiCode		:= 10000;
		tyInfoData.eSeverity	:= AlmSeverityInfo;
		tyInfoData.sAlmMsg		:= p_sInfoMsg;
	END_IF

	//Auto Reset
	fbDelayTm1(IN := bUpdateUIData , PT := T#2S); //Auto reset the Info Msg C0009 page. No need press.
	IF fbDelayTm1.Q = TRUE THEN

		//Clear Info Message
		tyInfoData.sProgNm		:= '';
		tyInfoData.udiCode		:= 0;
		tyInfoData.eSeverity	:= AlmSeverityNA;
		tyInfoData.sAlmMsg		:= '';

		bUpdateUIData  := FALSE;
		bFoundIndexUS1 := FALSE;
		bFoundIndexUS2 := FALSE;
		bFoundIndexUS3 := FALSE;
		bFoundIndexUS4 := FALSE;
		bFoundIndexDS1 := FALSE;
		bFoundIndexDS2 := FALSE;
		bFoundIndexDS3 := FALSE;
		bFoundIndexDS4 := FALSE;

		fbDelayTm1(IN := FALSE);
	END_IF

	//BatchId from Supervisory System
	sBatchId := tySendWorkOrderInfoAcc.tyData.sBatchId;

	//Retain sWorkOrderId for machine power cycle
	p_udiRetainDataAddr	:= ADR(sWorkOrderId);
	p_udiRetainDataLen	:= SIZEOF(sWorkOrderId);

	//Write Retain
//	IF EDGEPOS(bRcvWorkOrderInfo1) THEN
//    	sWorkOrderId := tySendWorkOrderInfoAcc.tyData.sWorkOrderId; //Receive from Svy
//		p_eAct := HermesActWriteRetain;

	IF EDGEPOS(bRetainNewAcc) THEN
    	sWorkOrderId := tySendWorkOrderInfoNewAcc.tyData.sWorkOrderId; //Receive from Svy
		p_eAct := HermesActWriteRetain;

	ELSIF EDGENEG(p_bSvyEn = TRUE) OR EDGENEG(p_bSvyPrep = TRUE) THEN
		sWorkOrderId := ''; //Empty if Supervisory Hermes disable
		p_eAct := HermesActWriteRetain;

	ELSIF EDGENEG(p_tyHermesConfiguration.tySvyParam.bFeatureQueryWorkOrderInfo = TRUE) THEN
		sWorkOrderId := ''; //Empty if no support
		p_eAct := HermesActWriteRetain;

	ELSIF EDGEPOS(p_bDeleteWorkOrder) THEN
		sWorkOrderId := ''; //Delete from UI
		tySendWorkOrderInfoNewAcc := tyDummySendWorkOrderInfoRcv;
		p_eAct := HermesActWriteRetain;
		p_bDeleteWorkOrder := FALSE;
	END_IF

	//Retain tySendWorkOrderInfoAcc (Loader Accept data)
	p_udiLoaderRetainDataAddr0	:= ADR(tySendWorkOrderInfoAcc);
	p_udiLoaderRetainDataLen0   := SIZEOF(tySendWorkOrderInfoAcc);

	//Retain tySendWorkOrderInfoNewAcc (Loader loaded Accept data)
	p_udiLoaderRetainDataAddr1	:= ADR(tySendWorkOrderInfoNewAcc);
	p_udiLoaderRetainDataLen1   := SIZEOF(tySendWorkOrderInfoNewAcc);

     //Retain tySendBypassWorkOrderInfoAcc (Bypass Accept data)
	p_udiBypassRetainDataAddr0	:= ADR(tySendBypassWorkOrderInfoAcc);
	p_udiBypassRetainDataLen0   := SIZEOF(tySendBypassWorkOrderInfoAcc);

	IF EDGEPOS (bRcvWorkOrderInfo1) THEN
		p_eAct := HermesActWriteRetainSendWO1;

	ELSIF EDGEPOS (bRetainNewAcc OR p_bDeleteWorkOrder) THEN
		p_eAct := HermesActWriteRetainSendWO2;

	ELSIF EDGEPOS (bRcvWorkBypassOrderInfo) THEN
		p_eAct := HermesActWriteRetainSendWO3;
	END_IF

	IF eStatus = Done AND eStat = HermesActWriteRetain THEN
		p_eAct		:= HermesActIdle;
	ELSIF eStatus = Done AND eStat = HermesActWriteRetainSendWO1 THEN
		p_eAct		:= HermesActIdle;
	ELSIF eStatus = Done AND eStat = HermesActWriteRetainSendWO2 THEN
		p_eAct		:= HermesActIdle;
	ELSIF eStatus = Done AND eStat = HermesActWriteRetainSendWO3 THEN
		p_eAct		:= HermesActIdle;
	END_IF

//	//Testing -> Read Retain
//	IF EDGEPOS(bTest) THEN
//		p_eAct := HermesActReadRetain;
//	END_IF
//
//	IF eStatus = Done AND eStat = HermesActReadRetain THEN
//		p_eAct		:= HermesActIdle;
//	END_IF

END_ACTION
```

#### Act_Background_QueryWorkOrderInfo.st
```iecst
(** 2021-08-01 **)
ACTION Act_Background_QueryWorkOrderInfo:

	IF eStatus2 <> Error THEN

//		IF EDGEPOS(p_bQueryWorkOrderInfo) AND p_bAcceptCondition THEN

//		IF (EDGEPOS((p_bSiemensMcModeChgPrep AND p_bOpsConvWaitForTopUpBrd OR (p_usiLinkProdRcpCurrRcpMcMod = 0 AND bQueryloaderWorkOrder = FALSE) AND bConnected AND p_bOpsRun) AND p_bQueryWorkOrderInfo = FALSE AND bManualQueryWO = FALSE(*AND p_bSiemensMcModeChgPrep = FALSE)*)  (*AND p_bAcceptCondition*) AND bReplyWorkOrderInfo= FALSE AND sWorkOrderId = ''))
//			 OR EDGEPOS (p_bQueryWorkOrderInfo) THEN        //Query For Loader           //ADD
		IF (EDGEPOS((p_bSiemensMcModeChgPrep AND (p_bOpsConvWaitForTopUpBrd OR p_usiLinkProdRcpCurrRcpMcMod = 0)  AND bQueryloaderWorkOrder = FALSE AND bConnected AND p_bOpsRun) AND p_bQueryWorkOrderInfo = FALSE AND bManualQueryWO = FALSE AND bReplyWorkOrderInfo= FALSE AND sWorkOrderId = ''))
			 OR EDGEPOS (p_bQueryWorkOrderInfo) THEN        //Query For Loader           //ADD

			fHermesAddOneMsgSend(ADR(a_eMsgSend) , ADR(udiMsgSendBffr) , HermesMsgTypeQueryWorkOrderInfo);

			fHermesGenerateUUID(ADR(tyQueryWorkOrderInfo.tyData.sQueryId) , p_tyDTStructure , pa_usiMacAddr); //Generate QueryID

			tyQueryWorkOrderInfo.tyData.sMachineId							:= p_sMcId;
			tyQueryWorkOrderInfo.tyData.sMagazineId							:= p_sMagazineId;
			tyQueryWorkOrderInfo.tyData.iSlotId								:= p_iSlotId;
			tyQueryWorkOrderInfo.tyData.sBarcode						    := p_sBarcode;

			tyQueryWorkOrderInfo.tyAvl.bQueryId							    := tyQueryWorkOrderInfo.tyData.sQueryId <> '';
			tyQueryWorkOrderInfo.tyAvl.bMachineId							:= tyQueryWorkOrderInfo.tyData.sMachineId <> '';
			tyQueryWorkOrderInfo.tyAvl.bMagazineId							:= tyQueryWorkOrderInfo.tyData.sMagazineId <> '';
			tyQueryWorkOrderInfo.tyAvl.bSlotId								:= tyQueryWorkOrderInfo.tyData.iSlotId <> 0;
			tyQueryWorkOrderInfo.tyAvl.bBarcode								:= tyQueryWorkOrderInfo.tyData.sBarcode <> '';

			bQueryloaderWorkOrder := TRUE;
			bRcvWorkOrderInfo1 := FALSE;                     //ADD
			bRcvWorkOrderInfo2 := FALSE;

		END_IF
		                                                                      //Reply Bypass Workorder
		IF EDGEPOS((p_bSiemensMcModeChgPrep AND bConnected AND p_bOpsRun) AND bReplyBypassWorkOrderInfo= FALSE AND p_bUSHermesUSRdy AND bNewIncomingBoard)  THEN        //Query For Bypass mode           //ADD

			fHermesAddOneMsgSend(ADR(a_eMsgSend) , ADR(udiMsgSendBffr) , HermesMsgTypeQueryBypassWOInfo);

			fHermesGenerateUUID(ADR(tyQueryBypassWorkOrderInfo.tyData.sQueryId) , p_tyDTStructure , pa_usiMacAddr); //Generate QueryID

			tyQueryBypassWorkOrderInfo.tyData.sMachineId							:= p_sMcId;
			tyQueryBypassWorkOrderInfo.tyData.sMagazineId							:= p_sMagazineId;
			tyQueryBypassWorkOrderInfo.tyData.iSlotId								:= p_iSlotId;
			tyQueryBypassWorkOrderInfo.tyData.sBarcode						        := sUSBarcode;

			tyQueryBypassWorkOrderInfo.tyAvl.bQueryId							    := tyQueryBypassWorkOrderInfo.tyData.sQueryId <> '';
			tyQueryBypassWorkOrderInfo.tyAvl.bMachineId						     	:= tyQueryBypassWorkOrderInfo.tyData.sMachineId <> '';
			tyQueryBypassWorkOrderInfo.tyAvl.bMagazineId							:= tyQueryBypassWorkOrderInfo.tyData.sMagazineId <> '';
			tyQueryBypassWorkOrderInfo.tyAvl.bSlotId								:= tyQueryBypassWorkOrderInfo.tyData.iSlotId <> 0;
			tyQueryBypassWorkOrderInfo.tyAvl.bBarcode								:= tyQueryBypassWorkOrderInfo.tyData.sBarcode <> '';

			bQueryBypassWorkOrder := TRUE;
			bRcvWorkBypassOrderInfo := FALSE;
			bRcvBypassWorkOrderInfo2 := FALSE;
			bRcvWorkOrderInfo3      :=FALSE;
		END_IF

		IF p_bQueryWorkOrderInfo AND p_bAcceptCondition =FALSE THEN
			bRstWorkOrderInfo := TRUE;
		END_IF

		IF tyMsgTypeRcv.bSendWorkOrderInfo THEN

//			IF p_bQueryWorkOrderInfo AND (udiStatus2 = 0) THEN //After CmpParamRcv
//			IF (p_bQueryWorkOrderInfo OR p_bOpsConvWaitForTopUpBrd) AND (udiStatus2 = 0) AND p_tyDI.bTopCoverSWSig THEN //After CmpParamRcv
			IF (p_bQueryWorkOrderInfo OR p_bSiemensMcModeChgPrep) AND (udiStatus2 = 0) THEN //After CmpParamRcv
				IF tySendWorkOrderInfoRcv.tyAvl.bWorkOrderId AND tySendWorkOrderInfoRcv.tyData.sWorkOrderId <> '' AND
				   tySendWorkOrderInfoRcv.tyData.rWidth >= 50.0 AND tySendWorkOrderInfoRcv.tyData.rWidth <= 460.0	(*AND p_bAcceptCondition*) THEN //Wait Accept Conditon On

					bRcvWorkOrderInfo1 := TRUE;
					bRetainNewAcc      := FALSE;                            //ADD
					bQueryloaderWorkOrder := FALSE;
					tySendWorkOrderInfoAcc := tySendWorkOrderInfoRcv;
					tyMsgTypeRcv.bSendWorkOrderInfo := FALSE;
					sWorkOrderId := tySendWorkOrderInfoAcc.tyData.sWorkOrderId;

				ELSIF (tySendWorkOrderInfoRcv.tyAvl.bWorkOrderId = FALSE) OR tySendWorkOrderInfoRcv.tyData.sWorkOrderId = '' OR
					tySendWorkOrderInfoRcv.tyData.rWidth < 50.0 OR tySendWorkOrderInfoRcv.tyData.rWidth > 460.0  THEN
					bRcvWorkOrderInfo2 := TRUE;
					tyMsgTypeRcv.bSendWorkOrderInfo := FALSE;
				END_IF

			ELSIF p_bSiemensMcModeChgPrep AND (udiStatus5 = 0) THEN
				IF tySendWorkOrderInfoRcv.tyAvl.bWorkOrderId AND (tySendWorkOrderInfoRcv.tyData.sWorkOrderId = p_tyUSBoardAvailableRcv.tyData.sWorkOrderId OR tySendWorkOrderInfoRcv.tyData.sWorkOrderId = p_tyUSBoardForecastRcv.tyData.sWorkOrderId) AND
					tySendWorkOrderInfoRcv.tyAvl.bBatchId AND (tySendWorkOrderInfoRcv.tyData.sBatchId = p_tyUSBoardAvailableRcv.tyData.sBatchId OR tySendWorkOrderInfoRcv.tyData.sBatchId = p_tyUSBoardForecastRcv.tyData.sBatchId) AND
					tySendWorkOrderInfoRcv.tyAvl.bWidth AND (tySendWorkOrderInfoRcv.tyData.rWidth = p_tyUSBoardAvailableRcv.tyData.rWidth OR tySendWorkOrderInfoRcv.tyData.rWidth = p_tyUSBoardForecastRcv.tyData.rWidth) AND
					tySendWorkOrderInfoRcv.tyData.rWidth >= 50.0 AND tySendWorkOrderInfoRcv.tyData.rWidth <= 460.0 THEN
					bRcvWorkBypassOrderInfo := TRUE;
					tySendBypassWorkOrderInfoAcc := tySendWorkOrderInfoRcv;
					tyMsgTypeRcv.bSendWorkOrderInfo := FALSE;
					bRcvWorkOrderInfo3      :=TRUE;
				ELSE
					bRcvBypassWorkOrderInfo2 := TRUE;
					tyMsgTypeRcv.bSendWorkOrderInfo := FALSE;
				END_IF

//			ELSIF p_bQueryWorkOrderInfo = FALSE  THEN
			ELSIF p_bQueryWorkOrderInfo = FALSE  AND p_bLinkDIPresentSen = FALSE AND ((udiStatus2 = 0) OR (udiStatus5 = 0)) THEN
				tyMsgTypeRcv.bSendWorkOrderInfo := FALSE;
			END_IF
		END_IF

		IF EDGEPOS (bRcvWorkOrderInfo1 = TRUE AND p_bAcceptCondition) THEN

			tyInfoData1.sProgNm		:= p_sProgNm;
			tyInfoData1.udiCode		:= 10000;
			tyInfoData1.eSeverity	:= AlmSeverityInfo;
			tyInfoData1.sAlmMsg		:= p_sInfoMsg1;

		ELSIF EDGEPOS( bRcvWorkOrderInfo2 = TRUE OR bRcvBypassWorkOrderInfo2) THEN

			tyInfoData2.sProgNm		:= p_sProgNm;
			tyInfoData2.udiCode		:= 10000;
			tyInfoData2.eSeverity	:= AlmSeverityInfo;
			tyInfoData2.sAlmMsg		:= p_sInfoMsg2;

//			bRcvWorkOrderInfo2      := FALSE;
//			bRcvBypassWorkOrderInfo2 := FALSE;

		ELSIF EDGEPOS (bRcvWorkOrderInfo1 = TRUE AND p_bAcceptCondition = FALSE) THEN
			tyInfoData4.sProgNm		:= p_sProgNm;
			tyInfoData4.udiCode		:= 10000;
			tyInfoData4.eSeverity	:= AlmSeverityInfo;
			tyInfoData4.sAlmMsg		:= p_sInfoMsg4;

		END_IF

		IF  bRstWorkOrderInfo = TRUE THEN

			tyInfoData3.sProgNm		:= p_sProgNm;
			tyInfoData3.udiCode		:= 10000;
			tyInfoData3.eSeverity	:= AlmSeverityInfo;
			tyInfoData3.sAlmMsg		:= p_sInfoMsg3;

		END_IF

		IF EDGEPOS (bRcvWorkOrderInfo1 OR bRcvWorkOrderInfo2) THEN                       //ReplyWorkOrderInfo for loader

			fHermesAddOneMsgSend(ADR(a_eMsgSend) , ADR(udiMsgSendBffr) , HermesMsgTypeReplyWorkOrderInfo);

			tyReplyWorkOrderInfo.tyData.sWorkOrderId					    := tySendWorkOrderInfoAcc.tyData.sWorkOrderId;
			tyReplyWorkOrderInfo.tyData.sBatchId					      	:= tySendWorkOrderInfoAcc.tyData.sBatchId;
		    IF p_bAcceptCondition AND bRcvWorkOrderInfo2 = FALSE AND p_usiLinkProdRcpCurrRcpMcMod =1  THEN
				tyReplyWorkOrderInfo.tyData.iStatus							    := 1;          //WorkOrder accepted
				bReplyWorkOrderInfo                                             := TRUE;
			ELSIF bRcvWorkOrderInfo2 THEN
				tyReplyWorkOrderInfo.tyData.iStatus							    := 0;         //WorkOrder Rejected
				bReplyWorkOrderInfo                                             := FALSE;
				bRcvWorkOrderInfo2                                              := FALSE;
			ELSE
				tyReplyWorkOrderInfo.tyData.iStatus							    := 2;          //WorkOrder accepted and queue
				bReplyWorkOrderInfo                                             := TRUE;
			END_IF

			tyReplyWorkOrderInfo.tyAvl.bWorkOrderId					:= tySendWorkOrderInfoAcc.tyData.sWorkOrderId <> '';
			tyReplyWorkOrderInfo.tyAvl.bBatchId                     := tySendWorkOrderInfoAcc.tyData.sBatchId <> '';
			tyReplyWorkOrderInfo.tyAvl.bStatus                      :=  TRUE;
		END_IF

		IF EDGEPOS (bRcvWorkOrderInfo3 OR bRcvBypassWorkOrderInfo2) THEN                       //ReplyWorkOrderInfo for Bypass
			fHermesAddOneMsgSend(ADR(a_eMsgSend) , ADR(udiMsgSendBffr) , HermesMsgTypeReplyWorkOrderInfo);

			tyReplyWorkOrderInfo.tyData.sWorkOrderId					    := tySendBypassWorkOrderInfoAcc.tyData.sWorkOrderId;
			tyReplyWorkOrderInfo.tyData.sBatchId					      	:= tySendBypassWorkOrderInfoAcc.tyData.sBatchId;

			IF p_bAcceptCondition AND p_usiLinkProdRcpCurrRcpMcMod =0 AND bRcvWorkOrderInfo3  THEN
				tyReplyWorkOrderInfo.tyData.iStatus							    := 1;          //WorkOrder accepted
				bReplyBypassWorkOrderInfo                                       := TRUE;
			ELSIF p_bAcceptCondition AND p_usiLinkProdRcpCurrRcpMcMod =1 AND bRcvWorkOrderInfo3 THEN
				tyReplyWorkOrderInfo.tyData.iStatus							    := 2;          //WorkOrder accepted and queue
				bReplyBypassWorkOrderInfo                                       := TRUE;
				bQueryBypassWorkOrder := FALSE;                                               //Add
			ELSIF bRcvBypassWorkOrderInfo2 THEN
				tyReplyWorkOrderInfo.tyData.iStatus							    := 0;          //WorkOrder Rejected
				bReplyBypassWorkOrderInfo                                       := TRUE;
				bRcvBypassWorkOrderInfo2                                        :=FALSE;
			END_IF
			tyReplyWorkOrderInfo.tyAvl.bWorkOrderId					:= tySendWorkOrderInfoAcc.tyData.sWorkOrderId <> '';
			tyReplyWorkOrderInfo.tyAvl.bBatchId                     := tySendWorkOrderInfoAcc.tyData.sBatchId <> '';
			tyReplyWorkOrderInfo.tyAvl.bStatus                      :=  TRUE;
		END_IF

		IF (*p_bSiemensMcModeChgPrep AND*) p_usiLinkProdRcpCurrRcpMcMod =1 AND  bReplyWorkOrderInfo AND p_bLinkDIPresentSen =FALSE AND p_tyDI.bConvLftSen = FALSE AND p_tyDI.bConvRgtSen = FALSE  AND p_bAcceptCondition AND p_bUITopUpBrdRdy = FALSE THEN  //AND p_tyDI.bTopCoverSWSig  //Add
			bClearWorkOrder := FALSE;
			tySendWorkOrderInfoNewAcc := tySendWorkOrderInfoAcc;
			diReqWidthInUM	:= REAL_TO_DINT(tySendWorkOrderInfoAcc.tyData.rWidth * 1000);
			p_tyProdRcpCurrRcp.diWidthInUM	:= diReqWidthInUM;
			diReqLoaderWidthInUM := diReqWidthInUM;                 //ADD
			bReplyWorkOrderInfo := FALSE;                           //ADD
			bRetainNewAcc := TRUE;                                  //ADD
//			bSendBoardForecast := TRUE;                             //ADD
		ELSIF (*p_bSiemensMcModeChgPrep AND*) p_usiLinkProdRcpCurrRcpMcMod =0 AND bReplyBypassWorkOrderInfo AND p_bAcceptCondition AND bNewIncomingBoard = FALSE THEN
//			tySendWorkOrderInfoNewAcc := tySendBypassWorkOrderInfoAcc;
			diReqWidthInUM	:= REAL_TO_DINT(tySendBypassWorkOrderInfoAcc.tyData.rWidth * 1000);
			IF p_eLinkMcParamUSCommMod = McSetCommModSMEMA THEN
				p_tyProdRcpCurrRcp.diWidthInUM := diReqLoaderWidthInUM;
			ELSE
				p_tyProdRcpCurrRcp.diWidthInUM	:= diReqWidthInUM;
			END_IF
			bQueryBypassWorkOrder := FALSE;
			bReplyBypassWorkOrderInfo := FALSE;
		END_IF

		IF (p_usiSelProdRcpStep = 1) THEN                         //Standby Bit
			bClearWorkOrder := TRUE;
		END_IF

	END_IF

	//		IF p_bQueryWorkOrderInfo = FALSE (*AND p_bLinkDIPresentSen*) AND p_bOpsConvWaitForTopUpBrd= FALSE THEN
	IF  (EDGEPOS(bRcvWorkOrderInfo1 = FALSE AND bRcvWorkOrderInfo2 = FALSE)) (*OR p_bOpsPneuTopUpBrdReq*) OR p_bOpsConvStepAllwTopUpBrd THEN
		//Clear Info Message 1
		tyInfoData1.sProgNm		:= '';
		tyInfoData1.udiCode		:= 0;
		tyInfoData1.eSeverity	:= AlmSeverityNA;
		tyInfoData1.sAlmMsg		:= '';
		bRcvWorkOrderInfo1 := FALSE;

		//Clear Info Message 2
		tyInfoData2.sProgNm		:= '';
		tyInfoData2.udiCode		:= 0;
		tyInfoData2.eSeverity	:= AlmSeverityNA;
		tyInfoData2.sAlmMsg		:= '';
		bRcvWorkOrderInfo2 := FALSE;

		//Clear Info Message 3
		tyInfoData3.sProgNm		:= '';
		tyInfoData3.udiCode		:= 0;
		tyInfoData3.eSeverity	:= AlmSeverityNA;
		tyInfoData3.sAlmMsg		:= '';
		bRstWorkOrderInfo := FALSE;

		//Clear Info Message 4
		tyInfoData4.sProgNm		:= '';
		tyInfoData4.udiCode		:= 0;
		tyInfoData4.eSeverity	:= AlmSeverityNA;
		tyInfoData4.sAlmMsg		:= '';
		bRcvWorkOrderInfo1 := FALSE;

	END_IF

	IF EDGEPOS ((*(p_bAcceptCondition AND*) p_bSiemensMcModeChgPrep AND ((p_bLinkStepStackMode )) AND p_bOpsConvWaitForTopUpBrd) AND p_usiLinkProdRcpCurrRcpMcMod =1 AND p_bUITopUpBrdRdy = FALSE AND p_bOpsConvTopUpBrdReq = FALSE  AND p_bOpsRun THEN //p_tyDI.bLoadPosSen OR   // AND p_tyDI.bBrdClrSen= FALSE AND p_tyDI.bBrdStackPresentSen = FALSE //Whenever lifter empty clear send work data
		tySendWorkOrderInfoNewAcc := tyDummySendWorkOrderInfoRcv;
		sWorkOrderId := '';
	END_IF

//	IF p_bSendBFId THEN                    //New changeover send Forecast one pulse only
//		bSendBoardForecast := FALSE;
//	END_IF

END_ACTION
```

#### Act_Background_SendBoardArrivedLane1.st
```iecst
(** 2021-08-01 **)
ACTION Act_Background_SendBoardArrivedLane1: //Send after our machine send out "StopTransport" message to upstream

	IF eStatus2 <> Error THEN
		IF tySServiceDescriptionRcv.tyData.tySupportedFeatures.bFeatureBoardTracking = TRUE AND p_tyParam.bFeatureBoardTracking AND bHandshakeDone THEN
			IF EDGEPOS(p_bUSHermesStopTransport1) THEN

				fHermesAddOneMsgSend(ADR(a_eMsgSend) , ADR(udiMsgSendBffr) , HermesMsgTypeBoardArrived1);

				tyBoardArrived1.tyData.sMachineId     	        := p_sMcId;
				tyBoardArrived1.tyData.iUpstreamLaneId    	    := p_tyHermesConfiguration.a_tyUSParam[0].iLaneID;
				tyBoardArrived1.tyData.sUpstreamInterfaceId     := p_tyHermesConfiguration.a_tyUSParam[0].sUpstreamInterfaceId;
				tyBoardArrived1.tyData.sMagazineId           	:= '';//sMagazineId;
				tyBoardArrived1.tyData.iSlotId     	            := 0;//iSlotId;
				tyBoardArrived1.tyData.eBoadTransfer    	    := p_eBoardTransfer1;//HermesTransferred;
				tyBoardArrived1.tyData.sBoardId     	        := p_tyUSBoardArrived1.tyData.sBoardId;
				tyBoardArrived1.tyData.sBoardIdCreatedBy     	:= p_tyUSBoardArrived1.tyData.sBoardIdCreatedBy;
				tyBoardArrived1.tyData.eFailedBoard				:= p_tyUSBoardArrived1.tyData.eFailedBoard;
				tyBoardArrived1.tyData.sProductTypeId			:= p_tyUSBoardArrived1.tyData.sProductTypeId;
				tyBoardArrived1.tyData.eFlippedBoard		  	:= p_tyUSBoardArrived1.tyData.eFlippedBoard;
				tyBoardArrived1.tyData.sTopBarcode				:= p_tyUSBoardArrived1.tyData.sTopBarcode;
				tyBoardArrived1.tyData.sBottomBarcode			:= p_tyUSBoardArrived1.tyData.sBottomBarcode;
				tyBoardArrived1.tyData.rLength					:= p_tyUSBoardArrived1.tyData.rLength;
				tyBoardArrived1.tyData.rWidth				    := p_tyUSBoardArrived1.tyData.rWidth;
				tyBoardArrived1.tyData.rThickness				:= p_tyUSBoardArrived1.tyData.rThickness;
				tyBoardArrived1.tyData.rConveyorSpeed		    := p_tyUSBoardArrived1.tyData.rConveyorSpeed;
				tyBoardArrived1.tyData.rTopClearanceHeight		:= p_tyUSBoardArrived1.tyData.rTopClearanceHeight;
				tyBoardArrived1.tyData.rBottomClearanceHeight	:= p_tyUSBoardArrived1.tyData.rBottomClearanceHeight;
				tyBoardArrived1.tyData.rWeight					:= p_tyUSBoardArrived1.tyData.rWeight;
				tyBoardArrived1.tyData.sWorkOrdedId             := p_tyUSBoardArrived1.tyData.sWorkOrderId;
				tyBoardArrived1.tyData.sBatchId                 := p_tyUSBoardArrived1.tyData.sBatchId;

			    tyBoardArrived1.tyAvl.bMachineId				:= tyBoardArrived1.tyData.sMachineId <> '';
		     	tyBoardArrived1.tyAvl.bUpstreamLaneId			:= tyBoardArrived1.tyData.iUpstreamLaneId <> 0;
		    	tyBoardArrived1.tyAvl.bUpstreamInterfaceId		:= tyBoardArrived1.tyData.sUpstreamInterfaceId <> '';
		    	tyBoardArrived1.tyAvl.bMagazineId		    	:= tyBoardArrived1.tyData.sMagazineId <> '';
		    	tyBoardArrived1.tyAvl.bSlotId				    := tyBoardArrived1.tyData.iSlotId <> 0;
		    	tyBoardArrived1.tyAvl.bBoardTransfer			:= TRUE;
				tyBoardArrived1.tyAvl.bBoardId					:= tyBoardArrived1.tyData.sBoardId <> '';
				tyBoardArrived1.tyAvl.bBoardIdCreatedBy			:= tyBoardArrived1.tyData.sBoardIdCreatedBy <> '';
				tyBoardArrived1.tyAvl.bFailedBoard				:= TRUE;
				tyBoardArrived1.tyAvl.bProductTypeId		  	:= tyBoardArrived1.tyData.sProductTypeId <> '';
				tyBoardArrived1.tyAvl.bFlippedBoard				:= TRUE;
				tyBoardArrived1.tyAvl.bTopBarcode			    := tyBoardArrived1.tyData.sTopBarcode <> '';
				tyBoardArrived1.tyAvl.bBottomBarcode		   	:= tyBoardArrived1.tyData.sBottomBarcode <> '';
				tyBoardArrived1.tyAvl.bLength				    := tyBoardArrived1.tyData.rLength <> 0;
				tyBoardArrived1.tyAvl.bWidth				  	:= (tyBoardArrived1.tyData.rWidth <> 0);
				tyBoardArrived1.tyAvl.bThickness			   	:= (tyBoardArrived1.tyData.rThickness <> 0);
				tyBoardArrived1.tyAvl.bConveyorSpeed		   	:= tyBoardArrived1.tyData.rConveyorSpeed <> 0;
				tyBoardArrived1.tyAvl.bTopClearanceHeight	    := (tyBoardArrived1.tyData.rTopClearanceHeight <> 0);
				tyBoardArrived1.tyAvl.bBottomClearanceHeight    := (tyBoardArrived1.tyData.rBottomClearanceHeight <> 0);
		    	tyBoardArrived1.tyAvl.bWeight				    := tyBoardArrived1.tyData.rWeight <> 0;
				tyBoardArrived1.tyAvl.bWorkOrderId				:= tyBoardArrived1.tyData.sWorkOrdedId <> '';
				tyBoardArrived1.tyAvl.bBatchId			    	:= tyBoardArrived1.tyData.sBatchId <> '';

			END_IF

		END_IF

	END_IF

END_ACTION
```

#### Act_Background_SendBoardDepartedLane1.st
```iecst
(** 2021-08-01 **)
ACTION Act_Background_SendBoardDepartedLane1: //Send after our machine send out "TransportFinished" message to downstream

	IF eStatus2 <> Error THEN
		IF tySServiceDescriptionRcv.tyData.tySupportedFeatures.bFeatureBoardTracking = TRUE AND p_tyParam.bFeatureBoardTracking AND bHandshakeDone THEN
			IF EDGEPOS(p_bDSHermesTransportFinished1) THEN

				fHermesAddOneMsgSend(ADR(a_eMsgSend) , ADR(udiMsgSendBffr) , HermesMsgTypeBoardDeparted1);

				tyBoardDeparted1.tyData.sMachineId     	        := p_sMcId;
				tyBoardDeparted1.tyData.iDownstreamLaneId    	:= p_tyHermesConfiguration.a_tyUSParam[0].iLaneID; //changed
				tyBoardDeparted1.tyData.sDownstreamInterfaceId  := p_tyHermesConfiguration.a_tyUSParam[0].sUpstreamInterfaceId; //changed
				tyBoardDeparted1.tyData.sMagazineId           	:= sMagazineId;
				tyBoardDeparted1.tyData.iSlotId     	        := iSlotId;
				tyBoardDeparted1.tyData.eBoadTransfer    	    := p_eBoardTransfer1;
				tyBoardDeparted1.tyData.sBoardId     	        := p_tyDSBoardDeparted1.tyData.sBoardId;
				tyBoardDeparted1.tyData.sBoardIdCreatedBy     	:= p_tyDSBoardDeparted1.tyData.sBoardIdCreatedBy;
				tyBoardDeparted1.tyData.eFailedBoard			:= p_tyDSBoardDeparted1.tyData.eFailedBoard;
				tyBoardDeparted1.tyData.sProductTypeId			:= p_tyDSBoardDeparted1.tyData.sProductTypeId;
				tyBoardDeparted1.tyData.eFlippedBoard			:= p_tyDSBoardDeparted1.tyData.eFlippedBoard;
				tyBoardDeparted1.tyData.sTopBarcode				:= p_tyDSBoardDeparted1.tyData.sTopBarcode;
				tyBoardDeparted1.tyData.sBottomBarcode			:= p_tyDSBoardDeparted1.tyData.sBottomBarcode;
				tyBoardDeparted1.tyData.rLength					:= p_tyDSBoardDeparted1.tyData.rLength;
				tyBoardDeparted1.tyData.rWidth				    := p_tyDSBoardDeparted1.tyData.rWidth;
				tyBoardDeparted1.tyData.rThickness				:= p_tyDSBoardDeparted1.tyData.rThickness;
				tyBoardDeparted1.tyData.rConveyorSpeed		    := p_tyDSBoardDeparted1.tyData.rConveyorSpeed;
				tyBoardDeparted1.tyData.rTopClearanceHeight		:= p_tyDSBoardDeparted1.tyData.rTopClearanceHeight;
				tyBoardDeparted1.tyData.rBottomClearanceHeight	:= p_tyDSBoardDeparted1.tyData.rBottomClearanceHeight;
				tyBoardDeparted1.tyData.rWeight					:= p_tyDSBoardDeparted1.tyData.rWeight;
				tyBoardDeparted1.tyData.sWorkOrdedId            := p_tyDSBoardDeparted1.tyData.sWorkOrderId;
				tyBoardDeparted1.tyData.sBatchId                := p_tyDSBoardDeparted1.tyData.sBatchId;

				tyBoardDeparted1.tyAvl.bMachineId				:= tyBoardDeparted1.tyData.sMachineId <> '';
				tyBoardDeparted1.tyAvl.bDownstreamLaneId		:= tyBoardDeparted1.tyData.iDownstreamLaneId <> 0;
				tyBoardDeparted1.tyAvl.bDownstreamInterfaceId	:= tyBoardDeparted1.tyData.sDownstreamInterfaceId <> '';
				tyBoardDeparted1.tyAvl.bMagazineId		    	:= tyBoardDeparted1.tyData.sMagazineId <> '';
				tyBoardDeparted1.tyAvl.bSlotId				    := tyBoardDeparted1.tyData.iSlotId <> 0;
				tyBoardDeparted1.tyAvl.bBoardTransfer		    := TRUE;
				tyBoardDeparted1.tyAvl.bBoardId					:= tyBoardDeparted1.tyData.sBoardId <> '';
				tyBoardDeparted1.tyAvl.bBoardIdCreatedBy		:= tyBoardDeparted1.tyData.sBoardIdCreatedBy <> '';
				tyBoardDeparted1.tyAvl.bFailedBoard				:= TRUE;
				tyBoardDeparted1.tyAvl.bProductTypeId		   	:= tyBoardDeparted1.tyData.sProductTypeId <> '';
				tyBoardDeparted1.tyAvl.bFlippedBoard			:= TRUE;
				tyBoardDeparted1.tyAvl.bTopBarcode			    := tyBoardDeparted1.tyData.sTopBarcode <> '';
				tyBoardDeparted1.tyAvl.bBottomBarcode		    := tyBoardDeparted1.tyData.sBottomBarcode <> '';
				tyBoardDeparted1.tyAvl.bLength				    := tyBoardDeparted1.tyData.rLength <> 0;
				tyBoardDeparted1.tyAvl.bWidth				    := (tyBoardDeparted1.tyData.rWidth <> 0);
				tyBoardDeparted1.tyAvl.bThickness			    := (tyBoardDeparted1.tyData.rThickness <> 0);
				tyBoardDeparted1.tyAvl.bConveyorSpeed		    := tyBoardDeparted1.tyData.rConveyorSpeed <> 0;
				tyBoardDeparted1.tyAvl.bTopClearanceHeight	    := (tyBoardDeparted1.tyData.rTopClearanceHeight <> 0);
				tyBoardDeparted1.tyAvl.bBottomClearanceHeight	:= (tyBoardDeparted1.tyData.rBottomClearanceHeight <> 0);
				tyBoardDeparted1.tyAvl.bWeight				    := tyBoardDeparted1.tyData.rWeight <> 0;
				tyBoardDeparted1.tyAvl.bWorkOrderId				:= tyBoardDeparted1.tyData.sWorkOrdedId <> '';
				tyBoardDeparted1.tyAvl.bBatchId			    	:= tyBoardDeparted1.tyData.sBatchId <> '';

			END_IF

		END_IF

	END_IF

END_ACTION
```

#### Act_Background_TCPSend.st
```iecst
(** 2021-08-01 **)
ACTION Act_Background_TCPSend:

	//Message Send (Generate XML Message)
	IF a_eMsgSend[0] <> HermesMsgTypeNA THEN

		IF a_eMsgSend[0] = HermesMsgTypeCheckAlive THEN
			fHermesFormCheckAlive(ADR(a_tyXMLTableDataSnd) , p_tyDTStructure , tyCheckAliveSnd);
			fTableConvertToXML(ADR(sSnd) , ADR(udiSndMsgLen) , SIZEOF(sSnd) , ADR(a_tyXMLTableDataSnd) , ADR(a_tyXMLTableDataSnd[0].sTitle) , ADR(a_tyXMLTableDataSnd[0].sValue) , ADR(a_tyXMLTableDataSnd[0].uiSize) , SIZEOF(a_tyXMLTableDataSnd[0]) , 12);

		ELSIF a_eMsgSend[0] = HermesMsgTypeCheckAlivePing THEN
			fHermesFormCheckAlive(ADR(a_tyXMLTableDataSnd) , p_tyDTStructure , tyCheckAlivePingSnd);
			fTableConvertToXML(ADR(sSnd) , ADR(udiSndMsgLen) , SIZEOF(sSnd) , ADR(a_tyXMLTableDataSnd) , ADR(a_tyXMLTableDataSnd[0].sTitle) , ADR(a_tyXMLTableDataSnd[0].sValue) , ADR(a_tyXMLTableDataSnd[0].uiSize) , SIZEOF(a_tyXMLTableDataSnd[0]) , 12);

		ELSIF a_eMsgSend[0] = HermesMsgTypeCheckAlivePong THEN
			fHermesFormCheckAlive(ADR(a_tyXMLTableDataSnd) , p_tyDTStructure , tyCheckAlivePongSnd);
			fTableConvertToXML(ADR(sSnd) , ADR(udiSndMsgLen) , SIZEOF(sSnd) , ADR(a_tyXMLTableDataSnd) , ADR(a_tyXMLTableDataSnd[0].sTitle) , ADR(a_tyXMLTableDataSnd[0].sValue) , ADR(a_tyXMLTableDataSnd[0].uiSize) , SIZEOF(a_tyXMLTableDataSnd[0]) , 12);

		ELSIF a_eMsgSend[0] = HermesMsgTypeSServiceDescription THEN
			fHermesFormSServiceDescription(ADR(a_tyXMLTableDataSnd) , p_tyDTStructure , tySServiceDescriptionSnd);
			fTableConvertToXML(ADR(sSnd) , ADR(udiSndMsgLen) , SIZEOF(sSnd) , ADR(a_tyXMLTableDataSnd) , ADR(a_tyXMLTableDataSnd[0].sTitle) , ADR(a_tyXMLTableDataSnd[0].sValue) , ADR(a_tyXMLTableDataSnd[0].uiSize) , SIZEOF(a_tyXMLTableDataSnd[0]) ,30);

		ELSIF a_eMsgSend[0] = HermesMsgTypeNotification THEN
			fHermesFormNotification(ADR(a_tyXMLTableDataSnd) , p_tyDTStructure , tyNotificationSnd);
			fTableConvertToXML(ADR(sSnd) , ADR(udiSndMsgLen) , SIZEOF(sSnd) , ADR(a_tyXMLTableDataSnd) , ADR(a_tyXMLTableDataSnd[0].sTitle) , ADR(a_tyXMLTableDataSnd[0].sValue) , ADR(a_tyXMLTableDataSnd[0].uiSize) , SIZEOF(a_tyXMLTableDataSnd[0]) , 14);

		ELSIF a_eMsgSend[0] = HermesMsgTypeBoardAvailable THEN
			eStatus1	:= Error;
			udiStatus1	:= 10125;	//Board Available Request To Send From Supervisory Hermes

		ELSIF a_eMsgSend[0] = HermesMsgTypeRevokeBoardAvl THEN
			eStatus1	:= Error;
			udiStatus1	:= 10122;	//Revoke Board Available Request To Send From Supervisory Hermes

		ELSIF a_eMsgSend[0] = HermesMsgTypeMachineReady THEN
			eStatus1	:= Error;
			udiStatus1	:= 10135;	//Machine Ready Request To Send From Supervisory Hermes

		ELSIF a_eMsgSend[0] = HermesMsgTypeRevokeMachineReady THEN
			eStatus1	:= Error;
			udiStatus1	:= 10136;	//Revoke Machine Ready Request To Send From Supervisory Hermes

		ELSIF a_eMsgSend[0] = HermesMsgTypeStartTransport THEN
			eStatus1	:= Error;
			udiStatus1	:= 10137;	//Start Transport Request To Send From Supervisory Hermes

		ELSIF a_eMsgSend[0] = HermesMsgTypeStopTransport THEN
			eStatus1	:= Error;
			udiStatus1	:= 10123;	//Stop Transport Request To Send From Supervisory Hermes

		ELSIF a_eMsgSend[0] = HermesMsgTypeTransportFinished THEN
			eStatus1	:= Error;
			udiStatus1	:= 10124;	//Transport Finished Request To Send From Supervisory Hermes

		ELSIF a_eMsgSend[0] = HermesMsgTypeSetConfiguration THEN
			eStatus1	:= Error;
			udiStatus1	:= 10138;	//Set Configuration Request To Send From Supervisory Hermes

		ELSIF a_eMsgSend[0] = HermesMsgTypeGetConfiguration THEN
			eStatus1	:= Error;
			udiStatus1	:= 10139;	//Get Configuration Request To Send From Supervisory Hermes

		ELSIF a_eMsgSend[0] = HermesMsgTypeCurrConfiguration THEN
			fHermesFormCurrentConfiguration(ADR(a_tyXMLTableDataSnd) , p_tyDTStructure , tyCurrentConfigurationSnd);
			fTableConvertToXML(ADR(sSnd) , ADR(udiSndMsgLen) , SIZEOF(sSnd) , ADR(a_tyXMLTableDataSnd) , ADR(a_tyXMLTableDataSnd[0].sTitle) , ADR(a_tyXMLTableDataSnd[0].sValue) , ADR(a_tyXMLTableDataSnd[0].uiSize) , SIZEOF(a_tyXMLTableDataSnd[0]) , 80);
			//10140

		ELSIF a_eMsgSend[0] = HermesMsgTypeBoardForecast THEN
			eStatus1	:= Error;
			udiStatus1	:= 10141;	//Board Forecast Request To Send From Supervisory Hermes

		ELSIF a_eMsgSend[0] = HermesMsgTypeQueryBoardInfo THEN
			eStatus1	:= Error;
			udiStatus1	:= 10142;	//Query Board Info Request To Send From Supervisory Hermes

		ELSIF a_eMsgSend[0] = HermesMsgTypeSendBoardInfo THEN
			eStatus1	:= Error;
			udiStatus1	:= 10159;	//Send Board Info Request To Send From Supervisory Hermes

	    ELSIF a_eMsgSend[0] = HermesMsgTypeQueryWorkOrderInfo THEN
	    	fHermesFormQueryWorkOrderInfo(ADR(a_tyXMLTableDataSnd) , p_tyDTStructure , tyQueryWorkOrderInfo);
		    fTableConvertToXML(ADR(sSnd) , ADR(udiSndMsgLen) , SIZEOF(sSnd) , ADR(a_tyXMLTableDataSnd) , ADR(a_tyXMLTableDataSnd[0].sTitle) , ADR(a_tyXMLTableDataSnd[0].sValue) , ADR(a_tyXMLTableDataSnd[0].uiSize) , SIZEOF(a_tyXMLTableDataSnd[0]) , 20);
			//10160

		ELSIF a_eMsgSend[0] = HermesMsgTypeQueryBypassWOInfo THEN
			fHermesFormQueryBypassWOInfo(ADR(a_tyXMLTableDataSnd) , p_tyDTStructure , tyQueryBypassWorkOrderInfo);
			fTableConvertToXML(ADR(sSnd) , ADR(udiSndMsgLen) , SIZEOF(sSnd) , ADR(a_tyXMLTableDataSnd) , ADR(a_tyXMLTableDataSnd[0].sTitle) , ADR(a_tyXMLTableDataSnd[0].sValue) , ADR(a_tyXMLTableDataSnd[0].uiSize) , SIZEOF(a_tyXMLTableDataSnd[0]) , 20);
			//10160

    	ELSIF a_eMsgSend[0] = HermesMsgTypeSendWorkOrderInfo THEN
	     	eStatus1	:= Error;
		    udiStatus1	:= 10161;	//Send Work Order Info Request To Send From Supervisory Hermes

	    ELSIF a_eMsgSend[0] = HermesMsgTypeBoardArrived1 THEN //Lane 1
		    fHermesFormBoardArrived(ADR(a_tyXMLTableDataSnd) , p_tyDTStructure , tyBoardArrived1);
		    fTableConvertToXML(ADR(sSnd) , ADR(udiSndMsgLen) , SIZEOF(sSnd) , ADR(a_tyXMLTableDataSnd) , ADR(a_tyXMLTableDataSnd[0].sTitle) , ADR(a_tyXMLTableDataSnd[0].sValue) , ADR(a_tyXMLTableDataSnd[0].uiSize) , SIZEOF(a_tyXMLTableDataSnd[0]) , 50);
			//10162

		ELSIF a_eMsgSend[0] = HermesMsgTypeBoardArrived2 THEN //Lane 2
			fHermesFormBoardArrived(ADR(a_tyXMLTableDataSnd) , p_tyDTStructure , tyBoardArrived2);
			fTableConvertToXML(ADR(sSnd) , ADR(udiSndMsgLen) , SIZEOF(sSnd) , ADR(a_tyXMLTableDataSnd) , ADR(a_tyXMLTableDataSnd[0].sTitle) , ADR(a_tyXMLTableDataSnd[0].sValue) , ADR(a_tyXMLTableDataSnd[0].uiSize) , SIZEOF(a_tyXMLTableDataSnd[0]) , 50);
			//10162

		ELSIF a_eMsgSend[0] = HermesMsgTypeBoardArrived3 THEN //Lane 3
			fHermesFormBoardArrived(ADR(a_tyXMLTableDataSnd) , p_tyDTStructure , tyBoardArrived3);
			fTableConvertToXML(ADR(sSnd) , ADR(udiSndMsgLen) , SIZEOF(sSnd) , ADR(a_tyXMLTableDataSnd) , ADR(a_tyXMLTableDataSnd[0].sTitle) , ADR(a_tyXMLTableDataSnd[0].sValue) , ADR(a_tyXMLTableDataSnd[0].uiSize) , SIZEOF(a_tyXMLTableDataSnd[0]) , 50);
			//10162

		ELSIF a_eMsgSend[0] = HermesMsgTypeBoardArrived4 THEN //Lane 4
			fHermesFormBoardArrived(ADR(a_tyXMLTableDataSnd) , p_tyDTStructure , tyBoardArrived4);
			fTableConvertToXML(ADR(sSnd) , ADR(udiSndMsgLen) , SIZEOF(sSnd) , ADR(a_tyXMLTableDataSnd) , ADR(a_tyXMLTableDataSnd[0].sTitle) , ADR(a_tyXMLTableDataSnd[0].sValue) , ADR(a_tyXMLTableDataSnd[0].uiSize) , SIZEOF(a_tyXMLTableDataSnd[0]) , 50);
			//10162

	    ELSIF a_eMsgSend[0] = HermesMsgTypeBoardDeparted1 THEN
	    	fHermesFormBoardDeparted(ADR(a_tyXMLTableDataSnd) , p_tyDTStructure , tyBoardDeparted1);
	    	fTableConvertToXML(ADR(sSnd) , ADR(udiSndMsgLen) , SIZEOF(sSnd) , ADR(a_tyXMLTableDataSnd) , ADR(a_tyXMLTableDataSnd[0].sTitle) , ADR(a_tyXMLTableDataSnd[0].sValue) , ADR(a_tyXMLTableDataSnd[0].uiSize) , SIZEOF(a_tyXMLTableDataSnd[0]) , 50);
			//10163

		ELSIF a_eMsgSend[0] = HermesMsgTypeBoardDeparted2 THEN
			fHermesFormBoardDeparted(ADR(a_tyXMLTableDataSnd) , p_tyDTStructure , tyBoardDeparted2);
			fTableConvertToXML(ADR(sSnd) , ADR(udiSndMsgLen) , SIZEOF(sSnd) , ADR(a_tyXMLTableDataSnd) , ADR(a_tyXMLTableDataSnd[0].sTitle) , ADR(a_tyXMLTableDataSnd[0].sValue) , ADR(a_tyXMLTableDataSnd[0].uiSize) , SIZEOF(a_tyXMLTableDataSnd[0]) , 50);
			//10163

		ELSIF a_eMsgSend[0] = HermesMsgTypeBoardDeparted3 THEN
			fHermesFormBoardDeparted(ADR(a_tyXMLTableDataSnd) , p_tyDTStructure , tyBoardDeparted3);
			fTableConvertToXML(ADR(sSnd) , ADR(udiSndMsgLen) , SIZEOF(sSnd) , ADR(a_tyXMLTableDataSnd) , ADR(a_tyXMLTableDataSnd[0].sTitle) , ADR(a_tyXMLTableDataSnd[0].sValue) , ADR(a_tyXMLTableDataSnd[0].uiSize) , SIZEOF(a_tyXMLTableDataSnd[0]) , 50);
			//10163

		ELSIF a_eMsgSend[0] = HermesMsgTypeBoardDeparted4 THEN
			fHermesFormBoardDeparted(ADR(a_tyXMLTableDataSnd) , p_tyDTStructure , tyBoardDeparted4);
			fTableConvertToXML(ADR(sSnd) , ADR(udiSndMsgLen) , SIZEOF(sSnd) , ADR(a_tyXMLTableDataSnd) , ADR(a_tyXMLTableDataSnd[0].sTitle) , ADR(a_tyXMLTableDataSnd[0].sValue) , ADR(a_tyXMLTableDataSnd[0].uiSize) , SIZEOF(a_tyXMLTableDataSnd[0]) , 50);
			//10163

		ELSIF a_eMsgSend[0] = HermesMsgTypeReplyWorkOrderInfo THEN
			fHermesFormReplyWorkOrderInfo(ADR(a_tyXMLTableDataSnd) , p_tyDTStructure , tyReplyWorkOrderInfo);
			fTableConvertToXML(ADR(sSnd) , ADR(udiSndMsgLen) , SIZEOF(sSnd) , ADR(a_tyXMLTableDataSnd) , ADR(a_tyXMLTableDataSnd[0].sTitle) , ADR(a_tyXMLTableDataSnd[0].sValue) , ADR(a_tyXMLTableDataSnd[0].uiSize) , SIZEOF(a_tyXMLTableDataSnd[0]) , 20);
			//10164    //ADD

		END_IF

		//Message Send
		IF p_bInternalUse = FALSE THEN
			fbSend.udiTCPIdent	:= udiClntIdent;
			fbSend.udiSndSize	:= udiSndMsgLen;
			fbSend(bEn := TRUE);
		ELSE
			sInternalSnd	:= sSnd;
		END_IF

		IF (fbSend.udiStatus = 0) OR (p_bInternalUse = TRUE) THEN

			fLogDTConvert(ADR(sDT) , p_dtCurrDT);
			memset(ADR(a_sLogList[udiLogCntr]) , 0 , SIZEOF(a_sLogList[udiLogCntr]));
			memcpy(ADR(a_sLogList[udiLogCntr]) + LEN(a_sLogList[udiLogCntr]) , ADR(sDT) , LEN(sDT));
			memcpy(ADR(a_sLogList[udiLogCntr]) + LEN(a_sLogList[udiLogCntr]) , ADR('$r$n') , LEN('$r$n'));
			memcpy(ADR(a_sLogList[udiLogCntr]) + LEN(a_sLogList[udiLogCntr]) , ADR('SND_TO_SVY$r$n') , LEN('SND_TO_SVY$r$n'));
			memcpy(ADR(a_sLogList[udiLogCntr]) + LEN(a_sLogList[udiLogCntr]) , ADR(sSnd) , LEN(sSnd));
			memcpy(ADR(a_sLogList[udiLogCntr]) + LEN(a_sLogList[udiLogCntr]) , ADR('$r$n$r$n') , LEN('$r$n$r$n'));

			udiLogCntr	:= udiLogCntr + 1;
			IF udiLogCntr = 11 THEN
				udiLogCntr	:= 1;
			END_IF

			Act_Background_NotificationSnd;
			fHermesRmvOneMsgSend(ADR(a_eMsgSend) , ADR(udiMsgSendBffr));

			fbSend(bEn := FALSE);

		ELSIF (fbSend.udiStatus = 2321) AND (p_bInternalUse = FALSE) THEN
			bRstConnection	:= TRUE;

		ELSIF (fbSend.udiStatus < 65534) AND (p_bInternalUse = FALSE) THEN
			eStatus1	:= Error;

			IF fbSend.udiStatus = 2300 THEN
				udiStatus1	:= 10143;	//Invalid Ident While Sending Data
			ELSIF fbSend.udiStatus = 2320 THEN
				udiStatus1	:= 10144;	//TCP Retry Send Data Error While Sending Data
			ELSIF fbSend.udiStatus = 2322 THEN
				udiStatus1	:= 10145;	//TCP Send Data Error
			ELSE
				udiStatus1	:= fbSend.udiStatus;
			END_IF

	    END_IF
	END_IF

END_ACTION
```

#### Act_InitGlobal.st
```iecst
(** 2021-08-01 **)
ACTION Act_InitGlobal:

	(* Always Change If Project Change *)

		//Digital Input
	p_tyDI ACCESS p_DI;

	//Pass Data To Link
	p_bLinkStartupRun ACCESS p_StartupRun;

	//Pass Data To Internal Use
	p_udiRstErr ACCESS p_RstErrReset;
	p_bPrep ACCESS p_NtParamHermesPrep;
	p_tyParam ACCESS p_HermesSvyParam;
	p_sIPAddr ACCESS p_HWInfoIPAddr;
	pa_usiMacAddr ACCESS p_HWInfoMacAddr;
	p_tyDTStructure ACCESS p_TimeCurrDTStruct;
	p_dtCurrDT ACCESS p_TimeCurrDT;
	p_sMcId ACCESS p_McParamMcNm;
	p_sRecipeNm ACCESS p_ProdRcpCurrRcp0Nm;

	//magazine id
	//p_sMagazineId ACCESS p_UIMagazineId;
	//p_iSlotId ACCESS p_UIMagazineSlotId;
	//p_sBarcode ACCESS p_UIPCBBarcode;

	p_udiAliveIdleTimeInSec ACCESS p_NtParamSvyHermesAliveTmInSec;
	p_tConnTimeOut ACCESS p_NtParamSvyHermesConnTO;
	p_diTransferInTO ACCESS p_McParamTranOutErrDlyTm;
	p_bNewBrdAvlLastZone ACCESS p_HermesBrdAvlDataNewBrdAvlLastZ;
	p_bOpsRun ACCESS p_OpsRun;
	p_udiFileKeepDay ACCESS p_NtParamSvyHermesFileKeepDay;
	p_sConfigFileName ACCESS p_NtParamSvyHermesConfigFileNm;
	p_sProgNm ACCESS p_NtParamSvyHermesProgNm;
	p_bNtSettingsLoadDone ACCESS p_StartupNtSettingsLoadDone;
	p_bSvyPrep ACCESS p_NtParamHermesSvyPrep;
	p_bSvyEn ACCESS p_McParamHermesSvyEn;
	p_bQueryWorkOrderInfo ACCESS p_UIQueryWorkOrderInfo;
	p_tyHermesConfiguration ACCESS p_HermesConfiguration;
	p_bUSHermesStopTransport1 ACCESS p_USHermesAStopTransportSnd; //Lane 1
	p_bUSHermesStopTransport2 ACCESS p_USHermesBStopTransportSnd; //Lane 2, open up for specific machine
//	p_bUSHermesStopTransport3 ACCESS p_USHermesStopTransportSnd3; //Lane 3, open up for specific machine
//	p_bUSHermesStopTransport4 ACCESS p_USHermesStopTransportSnd4; //Lane 4, open up for specific machine
	p_tyUSBoardArrived1 ACCESS p_USHermesABoardArrivedData; //Lane 1
	p_tyUSBoardArrived2 ACCESS p_USHermesBBoardArrivedData; //Lane 2, open up for specific machine
//	p_tyUSBoardArrived3 ACCESS p_USHermesBoardArrivedData3; //Lane 3, open up for specific machine
//	p_tyUSBoardArrived4 ACCESS p_USHermesBoardArrivedData4; //Lane 4, open up for specific machine

	p_bDSSMEMA1ConvStart ACCESS p_DSSMEMA1ConvStart;
	p_bDSSMEMA2ConvStart ACCESS p_DSSMEMA2ConvStart;
	p_bDSSMEMA3ConvStart ACCESS p_DSSMEMA3ConvStart;
//	p_bDSHermesTransportFinished1 ACCESS p_DSSMEMA1TransprtFinished; //p_DSHermesTransportFinishedSnd;
//	p_bDSHermesTransportFinished2 ACCESS p_DSSMEMA2TransprtFinished; //Lane 2, open up for specific machine
//	p_bDSHermesTransportFinished3 ACCESS p_DSSMEMA3TransprtFinished; //Lane 3, open up for specific machine
//	p_bDSHermesTransportFinished4 ACCESS p_DSHermesTransportFinishedSnd4; //Lane 4, open up for specific machine
//	p_tyDSBoardDeparted1 ACCESS p_DSHermesBoardDepartedData; //Lane 1
//	p_tyDSBoardDeparted2 ACCESS p_DSHermesBoardDepartedData2; //Lane 2, open up for specific machine
//	p_tyDSBoardDeparted3 ACCESS p_DSHermesBoardDepartedData3; //Lane 3, open up for specific machine
//	p_tyDSBoardDeparted4 ACCESS p_DSHermesBoardDepartedData4; //Lane 4, open up for specific machine
	p_eHermesStat ACCESS p_HermesStat;
	p_eHermesStatus ACCESS p_HermesStatus;
	p_eMcParamStat ACCESS p_McParamStat;
	p_eMcParamStatus ACCESS p_McParamStatus;
	//p_bAllZonesEmpty ACCESS p_DSHermesAllZonesEmpty; //All zones empty. Before empty, cannot change current sWorkOrderId.
	p_bDeleteWorkOrder ACCESS p_UIDeleteWorkOrder;
	p_bFirstMcIntheLine ACCESS p_NtParamHermesSvyFirstMc; //First machine in the line only can Query Work Order
	p_sRetainFileName ACCESS p_NtParamSvyHermesRetainFileNm;
	p_tyProdRcpCurrRcp ACCESS p_ProdRcpCurrRcp0;
	p_tyProdRcpCurrRcp1 ACCESS p_ProdRcpCurrRcp1;

	p_bSiemensMcModeChgPrep ACCESS p_McParamSiemensPrep;          //ADD   Include ReplyWorkOrderID & Machine mode changeover
	//p_bLinkDIPresentSen ACCESS p_DIBrdStackPresentSen;                     //ADD for Loader
	//p_bLinkOpsConvGdBrd	ACCESS
	//p_bOpsConvTopUpBrdReq ACCESS p_OpsConvTopUpBrdReq;
	//p_bOpsConvWaitForTopUpBrd ACCESS p_OpsConvWaitForTopUpBrd;
	//p_bUITopUpBrdRdy ACCESS p_UITopUpBrdRdy;
	//p_bSendBFId ACCESS p_SendBFId;
	p_usiSelProdRcpStep  ACCESS p_SelProdRcpStep;

	//p_bOpsPneuStepAllwInitConv ACCESS p_OpsPneuStepAllwInitConv;
	//p_bOpsConvStepChkInit ACCESS p_OpsConvStepChkInit;
	//p_bOpsPneuTopUpBrdReq ACCESS p_OpsPneuTopUpBrdReq;
	//p_bOpsConvStepAllwTopUpBrd ACCESS p_OpsConvStepAllwTopUpBrd;

	p_usiLinkProdRcpCurrRcpMcMod ACCESS p_ProdRcpCurrRcp0McMod;      //Add
	//p_bUSSMEMAUSRdy ACCESS p_USSMEMAUSRdy;
	p_bUSHermesUSRdy ACCESS p_USHermesAUSRdy;
	p_bLinkBrdAvlDataNewBrdAvl1stZ ACCESS p_HermesBrdAvlDataNewBrdAvl1stZ;
	pa_tyLinkXMLTableDataBrdAvl1 ACCESS p_HermesBrdAvlDataTable1stZ; //lane 1 B.A
	p_iLinkXMLTableDataBrdAvlTtlIdx1 ACCESS p_HermesBrdAvlDataTtlIdx1stZ; //lane 1 B.A
	//p_tyUSBoardAvailableRcv ACCESS  p_USBoardAvailableRcv;
	//p_tyUSBoardForecastRcv ACCESS p_USBoardForecastRcv;
	//p_bLoaderChangeOver ACCESS p_LoaderChangeOver;
	//p_bLinkStepStackMode ACCESS p_McParamStepStackMode;

	//p_eLinkMcParamUSCommMod ACCESS p_McParamUSCommMod;

	p_bOpsTravLifGdBrdChk ACCESS p_OpsTravLifWGdBrdChk;

	p_diBuffer1Slt ACCESS p_Buffer1SlotNo;
	p_diBuffer2Slt ACCESS p_Buffer2SlotNo;
	p_diBuffer3Slt ACCESS p_Buffer3SlotNo;

	p_bPshrConvHvBrd ACCESS p_PshrConvHvBrd;

	p_bUSHermesARcvBoardInfo ACCESS p_USHermesARcvBoardInfoOk;
	p_tyUSHermesSendBoardInfoAcpt ACCESS p_USHermesABoardInfoData;
	(* Always Change If Project Change *)
END_ACTION
```

#### Act_Initial.st
```iecst
(** 2021-08-01 **)
ACTION Act_Initial:

	//Initial
	sStatTxt	:= a_sStatText[eStat];

	fbCreateSvr.udiSndBffrSize		:= p_udiSndBffrSize;
	fbCreateSvr.udiRcvBffrSize		:= p_udiRcvBffrSize;
	fbCreateSvr.udiAliveIdleTmInSec	:= p_udiAliveIdleTimeInSec;
	fbCreateSvr(bEn := FALSE);

	fbListen(bEn := FALSE);

	fbRcv.udiBffrSize	:= SIZEOF(sRcv);
	fbRcv.p_BffrDest	:= ADR(sRcv);
	fbRcv(bEn := FALSE);

	fbSend.p_BffrDest	:= ADR(sSnd);
	fbSend(bEn := FALSE);

	fbCloseSvr(bEn := FALSE);
	fbCloseClnt(bEn := FALSE);

	fbParseXMLTable.p_XMLTable	:= ADR(a_tyXMLTableDataRcv);

	fbCheckAlive(bEn := FALSE);

	fbCheckAliveSendPing(bEn := FALSE);

	fbCheckAliveRcvPing(bEn := FALSE);

	fbSequenceSvy.p_tyMsgTypeRcv	:= ADR(tyMsgTypeRcv);
	fbSequenceSvy(bEn := FALSE);

	fbSequenceTO(bEn := FALSE);

	fbFileAppend1.sDevice	:= 'Log';
	fbFileAppend1(bEn := FALSE);

	fbFileOldDel1.sDevice			:= 'Log';
	fbFileOldDel1.sPath				:= '';
	fbFileOldDel1.sKeyword			:= p_sProgNm;
	fbFileOldDel1.udiFileKeepDay	:= p_udiFileKeepDay;
	fbFileOldDel1(bEn := FALSE);

	fbFileRead1.sDevice			:= 'Retain';
	fbFileRead1.sFile			:= p_sRetainFileName;
	fbFileRead1.udiOffset		:= 0;
	fbFileRead1(bEn := FALSE);

	fbFileWrite1.sDevice		:= 'Retain';
	fbFileWrite1.sFile			:= p_sRetainFileName;
	fbFileWrite1.udiOffset		:= 0;
	fbFileWrite1.udiOption		:= 0;
	fbFileWrite1(bEn := FALSE);

	fbFileRead2.sDevice			:= 'Retain';
	fbFileRead2.sFile			:= p_sRetainFileName1;
	fbFileRead2.udiOffset		:= 0;
	fbFileRead2(bEn := FALSE);

	fbFileWrite2.sDevice		:= 'Retain';
	fbFileWrite2.sFile			:= p_sRetainFileName1;
	fbFileWrite2.udiOffset		:= 0;
	fbFileWrite2.udiOption		:= 0;
	fbFileWrite2(bEn := FALSE);

	fbFileRead3.sDevice			:= 'Retain';
	fbFileRead3.sFile			:= p_sRetainFileName2;
	fbFileRead3.udiOffset		:= 0;
	fbFileRead3(bEn := FALSE);

	fbFileWrite3.sDevice		:= 'Retain';
	fbFileWrite3.sFile			:= p_sRetainFileName2;
	fbFileWrite3.udiOffset		:= 0;
	fbFileWrite3.udiOption		:= 0;
	fbFileWrite3(bEn := FALSE);

	fbFileRead4.sDevice			:= 'Retain';
	fbFileRead4.sFile			:= p_sRetainFileName3;
	fbFileRead4.udiOffset		:= 0;
	fbFileRead4(bEn := FALSE);

	fbFileWrite4.sDevice		:= 'Retain';
	fbFileWrite4.sFile			:= p_sRetainFileName3;
	fbFileWrite4.udiOffset		:= 0;
	fbFileWrite4.udiOption		:= 0;
	fbFileWrite4(bEn := FALSE);

	diReqLoaderWidthInUM := REAL_TO_DINT(tySendWorkOrderInfoAcc.tyData.rWidth * 1000);

END_ACTION
```

#### Act_InitLocal.st
```iecst
(** 2021-08-01 **)
ACTION Act_InitLocal:

	//Input Reference Link To Local Variable
	p_eAct ACCESS ADR(eAct);
	p_udiRstErr ACCESS ADR(udiRstErr);
	p_bPrep ACCESS ADR(bPrep);
	p_bEn ACCESS ADR(bEn);
	p_bDis ACCESS ADR(bDis);
	p_tyParam ACCESS ADR(tyParam);
	p_sIPAddr ACCESS ADR(sIPAddr);
	pa_usiMacAddr ACCESS ADR(a_usiMacAddr);
	p_tyDTStructure ACCESS ADR(tyDTStructure);
	p_dtCurrDT ACCESS ADR(dtCurrDT);
	p_sMcId ACCESS ADR(sMcId);
	p_sMagazineId ACCESS ADR(sMagazineId);
	p_iSlotId ACCESS ADR(iSlotId);
	p_eBoardTransfer1 ACCESS ADR(eBoardTransfer1);
	p_eBoardTransfer2 ACCESS ADR(eBoardTransfer2);
	p_eBoardTransfer3 ACCESS ADR(eBoardTransfer3);
	p_eBoardTransfer4 ACCESS ADR(eBoardTransfer4);
	p_sVersion ACCESS ADR(sVersion);
	p_sBarcode ACCESS ADR(sBarcode);
	p_sRecipeNm ACCESS ADR(sRecipeNm);
	p_udiSndBffrSize ACCESS ADR(udiSndBffrSize);
	p_udiRcvBffrSize ACCESS ADR(udiRcvBffrSize);
	p_udiAliveIdleTimeInSec ACCESS ADR(udiAliveIdleTimeInSec);
	p_tConnTimeOut ACCESS ADR(tConnTimeOut);
	p_diTransferInTO ACCESS ADR(diTransferInTO);
	p_bNewBrdAvlLastZone ACCESS ADR(bNewBrdAvl);
	p_bOpsRun ACCESS ADR(bOpsRun);
	p_udiFileKeepDay ACCESS ADR(udiFileKeepDay);
	p_sConfigFileName ACCESS ADR(sConfigFileName);
	p_sProgNm ACCESS ADR(sProgNm);
	p_bNtSettingsLoadDone ACCESS ADR(bNtSettingsLoadDone);
	p_bSvyPrep ACCESS ADR(bSvyPrep);
	p_bSvyEn ACCESS ADR(bSvyEn);
	p_bQueryWorkOrderInfo ACCESS ADR(bQueryWorkOrderInfo);
	p_tyHermesConfiguration ACCESS ADR(tyHermesCurrConfiguration);
	p_bUSHermesStopTransport1 ACCESS ADR(bUSHermesStopTransportSnd1); //Lane 1
	p_bUSHermesStopTransport2 ACCESS ADR(bUSHermesStopTransportSnd2); //Lane 2
	p_bUSHermesStopTransport3 ACCESS ADR(bUSHermesStopTransportSnd3); //Lane 3
	p_bUSHermesStopTransport4 ACCESS ADR(bUSHermesStopTransportSnd4); //Lane 4
	p_tyUSBoardArrived1 ACCESS ADR(tyUSHermesBoardArrivedData1); //Lane 1
	p_tyUSBoardArrived2 ACCESS ADR(tyUSHermesBoardArrivedData2); //Lane 2
	p_tyUSBoardArrived3 ACCESS ADR(tyUSHermesBoardArrivedData3); //Lane 3
	p_tyUSBoardArrived4 ACCESS ADR(tyUSHermesBoardArrivedData4); //Lane 4
	p_bDSHermesTransportFinished1 ACCESS ADR(bDSHermesTransportFinishedSnd1); //Lane 1
	p_bDSHermesTransportFinished2 ACCESS ADR(bDSHermesTransportFinishedSnd2); //Lane 2
	p_bDSHermesTransportFinished3 ACCESS ADR(bDSHermesTransportFinishedSnd3); //Lane 3
	p_bDSHermesTransportFinished4 ACCESS ADR(bDSHermesTransportFinishedSnd4); //Lane 4
	p_tyDSBoardDeparted1 ACCESS ADR(tyDSHermesBoardDepartedData1); //Lane 1
	p_tyDSBoardDeparted2 ACCESS ADR(tyDSHermesBoardDepartedData2); //Lane 2
	p_tyDSBoardDeparted3 ACCESS ADR(tyDSHermesBoardDepartedData3); //Lane 3
	p_tyDSBoardDeparted4 ACCESS ADR(tyDSHermesBoardDepartedData4); //Lane 4
	p_sInfoMsg ACCESS ADR(sInfoMsg);
	p_sInfoMsg1 ACCESS ADR(sInfoMsg1);
	p_sInfoMsg2 ACCESS ADR(sInfoMsg2);
	p_sInfoMsg3 ACCESS ADR(sInfoMsg3);
	p_sInfoMsg4 ACCESS ADR(sInfoMsg4);
	p_bInternalUse ACCESS ADR(bInternalUse);
	p_sInternalRcv ACCESS ADR(sInternalRcv);
	p_bAcceptCondition ACCESS ADR(bAcceptCondition);
	p_bAllZonesEmpty ACCESS ADR(bAllZonesEmpty);
	p_bDeleteWorkOrder ACCESS ADR(bDeleteWorkOrder);
	p_bFirstMcIntheLine ACCESS ADR(bFirstMcIntheLine);
	p_sRetainFileName ACCESS ADR(sRetainFileName);
	p_udiRetainDataAddr ACCESS ADR(udiRetainDataAddr);
	p_udiRetainDataLen ACCESS ADR(udiRetainDataLen);
	p_sRetainFileName1 ACCESS ADR(sRetainFileName1);           //ADD
	p_sRetainFileName2 ACCESS ADR(sRetainFileName2);
	p_sRetainFileName3 ACCESS ADR(sRetainFileName3);
	p_udiLoaderRetainDataAddr0 ACCESS ADR(udiLoaderRetainDataAddr0);
	p_udiLoaderRetainDataLen0 ACCESS ADR(udiLoaderRetainDataLen0);
	p_udiLoaderRetainDataAddr1 ACCESS ADR(udiLoaderRetainDataAddr1);
	p_udiLoaderRetainDataLen1 ACCESS ADR(udiLoaderRetainDataLen1);
	p_udiBypassRetainDataAddr0 ACCESS ADR(udiBypassRetainDataAddr0);
	p_udiBypassRetainDataLen0 ACCESS ADR(udiBypassRetainDataLen0);        //ADD

	p_tyUSBoardAvailableRcv ACCESS ADR(tyHermesBARcv);
	p_tyUSBoardForecastRcv ACCESS ADR(tyHermesBFRcv);
	p_bOpsConvWaitForTopUpBrd ACCESS ADR(bOpsConvWaitForTopUpBrd);
	p_bUITopUpBrdRdy ACCESS	ADR(bUITopUpBrdRdy);	//Mag Present Sensor
	p_bLinkDIPresentSen ACCESS ADR(bDIPresentSen);  //Potential for query 3 empty Magzine Work Order
	p_bOpsConvStepAllwTopUpBrd ACCESS ADR(bOpsConvStepAllwTopUpBrd);
	p_bOpsConvTopUpBrdReq ACCESS ADR(bOpsConvTopUpBrdReq);
	p_bLinkStepStackMode ACCESS ADR(bLinkStepStackMode);
END_ACTION
```
